Yaskawa INFORM job: u_tourne4TRJ0.JBI

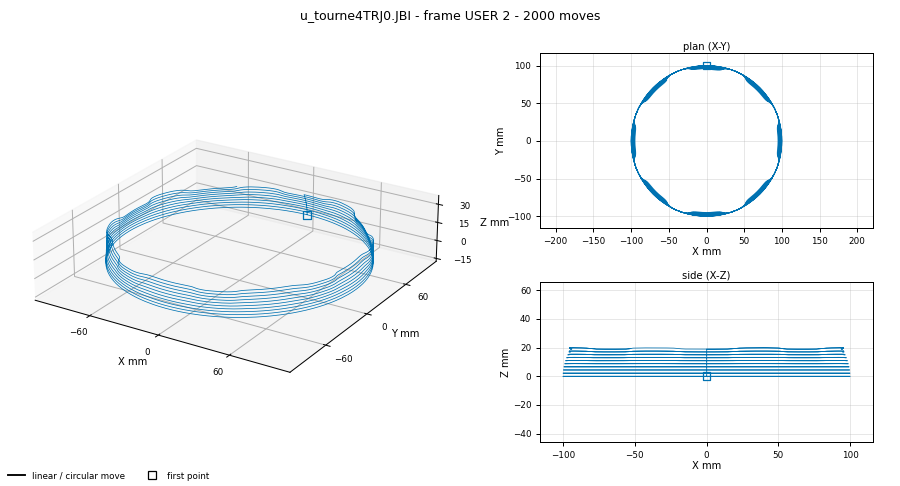
[picture p0: tool path of u_tourne4TRJ0.JBI in frame USER 2, 2000 of 2000 moves have a stored position in this frame; points joined in program order, loops and branches not executed]
/JOB
//NAME u_tourne4TRJ0
///FOLDERNAME DEMO
//POS
///NPOS 2000,0,2000,0,0,0
///USER 2
///TOOL 7
///POSTYPE USER
///RECTAN
///RCONF 1,0,0,0,0,0,0,0,0,0,0,0,0,0,0,0,0,0,0,0,0,0,0,0
C00000=0.000,100.000,0.000,-180.0000,0.0000,-90.0000
C00001=5.792,99.832,0.000,-180.0000,0.0000,-93.3204
C00002=10.988,99.394,0.000,-180.0000,0.0000,-96.3084
C00003=15.564,98.781,0.000,-180.0000,0.0000,-98.9540
C00004=18.698,98.237,0.000,-180.0000,0.0000,-100.7765
C00005=20.854,97.801,0.000,-180.0000,0.0000,-102.0369
C00006=22.593,97.414,0.000,-180.0000,0.0000,-103.0576
C00007=24.351,96.990,0.000,-180.0000,0.0000,-104.0938
C00008=26.550,96.411,0.000,-180.0000,0.0000,-105.3967
C00009=29.248,95.627,0.000,-180.0000,0.0000,-107.0065
C00010=32.094,94.710,0.000,-180.0000,0.0000,-108.7198
C00011=34.739,93.772,0.000,-180.0000,0.0000,-110.3278
C00012=37.121,92.855,0.000,-180.0000,0.0000,-111.7902
C00013=39.410,91.907,0.000,-180.0000,0.0000,-113.2098
C00014=41.743,90.871,0.000,-180.0000,0.0000,-114.6724
C00015=44.276,89.664,0.000,-180.0000,-0.0000,-116.2801
C00016=46.937,88.300,0.000,-180.0000,-0.0000,-117.9935
C00017=49.400,86.946,0.000,-180.0000,0.0000,-119.6039
C00018=51.363,85.801,0.000,-180.0000,0.0000,-120.9060
C00019=52.906,84.858,0.000,-180.0000,0.0000,-121.9421
C00020=54.410,83.902,0.000,-180.0000,0.0000,-122.9632
C00021=56.242,82.685,0.000,-180.0000,0.0000,-124.2234
C00022=58.844,80.854,0.000,-180.0000,0.0000,-126.0464
C00023=62.512,78.053,0.000,-180.0000,0.0000,-128.6909
C00024=66.496,74.687,0.000,-180.0000,0.0000,-131.6796
C00025=70.711,70.711,0.000,-180.0000,0.0000,-135.0000
C00026=74.687,66.496,0.000,-180.0000,0.0000,-138.3204
C00027=78.053,62.512,0.000,-180.0000,0.0000,-141.3091
C00028=80.854,58.844,0.000,-180.0000,-0.0000,-143.9536
C00029=82.685,56.242,0.000,-180.0000,0.0000,-145.7766
C00030=83.902,54.410,0.000,-180.0000,0.0000,-147.0368
C00031=84.858,52.906,0.000,-180.0000,0.0000,-148.0579
C00032=85.801,51.363,0.000,-180.0000,0.0000,-149.0940
C00033=86.946,49.400,0.000,-180.0000,0.0000,-150.3961
C00034=88.300,46.937,0.000,-180.0000,0.0000,-152.0065
C00035=89.664,44.276,0.000,-180.0000,0.0000,-153.7199
C00036=90.871,41.743,0.000,-180.0000,0.0000,-155.3276
C00037=91.907,39.410,0.000,-180.0000,0.0000,-156.7902
C00038=92.855,37.121,0.000,-180.0000,0.0000,-158.2098
C00039=93.772,34.739,0.000,-180.0000,0.0000,-159.6722
C00040=94.710,32.094,0.000,-180.0000,0.0000,-161.2802
C00041=95.627,29.248,0.000,-180.0000,0.0000,-162.9935
C00042=96.411,26.550,0.000,-180.0000,0.0000,-164.6033
C00043=96.990,24.351,0.000,-180.0000,0.0000,-165.9062
C00044=97.414,22.593,0.000,-180.0000,0.0000,-166.9424
C00045=97.801,20.854,0.000,-180.0000,0.0000,-167.9631
C00046=98.237,18.698,0.000,-180.0000,0.0000,-169.2235
C00047=98.781,15.564,0.000,-180.0000,0.0000,-171.0460
C00048=99.394,10.988,0.000,-180.0000,0.0000,-173.6916
C00049=99.832,5.792,0.000,-180.0000,0.0000,-176.6796
C00050=100.000,0.000,0.000,-180.0000,0.0000,-180.0000
C00051=99.832,-5.792,0.000,-180.0000,0.0000,-183.3204
C00052=99.394,-10.988,0.000,-180.0000,0.0000,-186.3084
C00053=98.781,-15.564,0.000,-180.0000,0.0000,-188.9540
C00054=98.237,-18.698,0.000,-180.0000,0.0000,-190.7765
C00055=97.801,-20.854,0.000,-180.0000,0.0000,-192.0369
C00056=97.414,-22.593,0.000,-180.0000,0.0000,-193.0576
C00057=96.990,-24.351,0.000,-180.0000,0.0000,-194.0938
C00058=96.411,-26.550,0.000,-180.0000,0.0000,-195.3967
C00059=95.627,-29.248,0.000,-180.0000,0.0000,-197.0065
C00060=94.710,-32.094,0.000,-180.0000,0.0000,-198.7198
C00061=93.772,-34.739,0.000,-180.0000,0.0000,-200.3278
C00062=92.855,-37.121,0.000,-180.0000,0.0000,-201.7902
C00063=91.907,-39.410,0.000,-180.0000,0.0000,-203.2098
C00064=90.871,-41.743,0.000,-180.0000,0.0000,-204.6724
C00065=89.664,-44.276,0.000,-180.0000,0.0000,-206.2801
C00066=88.300,-46.937,0.000,-180.0000,0.0000,-207.9935
C00067=86.946,-49.400,0.000,-180.0000,0.0000,-209.6039
C00068=85.801,-51.363,0.000,-180.0000,0.0000,-210.9060
C00069=84.858,-52.906,0.000,-180.0000,0.0000,-211.9421
C00070=83.902,-54.410,0.000,-180.0000,0.0000,-212.9632
C00071=82.685,-56.242,0.000,-180.0000,0.0000,-214.2234
C00072=80.854,-58.844,0.000,-180.0000,0.0000,-216.0464
C00073=78.053,-62.512,0.000,-180.0000,0.0000,-218.6909
C00074=74.687,-66.496,0.000,-180.0000,0.0000,-221.6796
C00075=70.711,-70.711,0.000,-180.0000,0.0000,-225.0000
C00076=66.496,-74.687,0.000,-180.0000,0.0000,-228.3204
C00077=62.512,-78.053,0.000,-180.0000,0.0000,-231.3091
C00078=58.844,-80.854,0.000,-180.0000,0.0000,-233.9536
C00079=56.242,-82.685,0.000,-180.0000,0.0000,-235.7766
C00080=54.410,-83.902,0.000,-180.0000,0.0000,-237.0368
C00081=52.906,-84.858,0.000,-180.0000,0.0000,-238.0579
C00082=51.363,-85.801,0.000,-180.0000,0.0000,-239.0940
C00083=49.400,-86.946,0.000,-180.0000,-0.0000,-240.3961
C00084=46.937,-88.300,0.000,-180.0000,0.0000,-242.0065
C00085=44.276,-89.664,0.000,-180.0000,0.0000,-243.7199
C00086=41.743,-90.871,0.000,-180.0000,0.0000,-245.3276
C00087=39.410,-91.907,0.000,-180.0000,0.0000,-246.7902
C00088=37.121,-92.855,0.000,-180.0000,0.0000,-248.2098
C00089=34.739,-93.772,0.000,-180.0000,0.0000,-249.6722
C00090=32.094,-94.710,0.000,-180.0000,0.0000,-251.2802
C00091=29.248,-95.627,0.000,-180.0000,0.0000,-252.9935
C00092=26.550,-96.411,0.000,-180.0000,0.0000,-254.6033
C00093=24.351,-96.990,0.000,-180.0000,0.0000,-255.9062
C00094=22.593,-97.414,0.000,-180.0000,0.0000,-256.9424
C00095=20.854,-97.801,0.000,-180.0000,0.0000,-257.9631
C00096=18.698,-98.237,0.000,-180.0000,0.0000,-259.2235
C00097=15.564,-98.781,0.000,-180.0000,0.0000,-261.0460
C00098=10.988,-99.394,0.000,-180.0000,0.0000,-263.6916
C00099=5.792,-99.832,0.000,-180.0000,0.0000,-266.6796
C00100=0.000,-100.000,0.000,180.0000,-0.0000,-270.0000
C00101=0.000,-100.000,0.000,180.0000,-0.0000,-270.0000
C00102=-5.792,-99.832,0.000,-180.0000,-0.0000,-273.3204
C00103=-10.988,-99.394,0.000,-180.0000,-0.0000,-276.3084
C00104=-15.564,-98.781,0.000,-180.0000,-0.0000,-278.9540
C00105=-18.698,-98.237,0.000,-180.0000,-0.0000,-280.7765
C00106=-20.854,-97.801,0.000,-180.0000,-0.0000,-282.0369
C00107=-22.593,-97.414,0.000,-180.0000,-0.0000,-283.0576
C00108=-24.351,-96.990,0.000,-180.0000,-0.0000,-284.0938
C00109=-26.550,-96.411,0.000,-180.0000,-0.0000,-285.3967
C00110=-29.248,-95.627,0.000,-180.0000,-0.0000,-287.0065
C00111=-32.094,-94.710,0.000,-180.0000,-0.0000,-288.7198
C00112=-34.739,-93.772,0.000,-180.0000,-0.0000,-290.3278
C00113=-37.121,-92.855,0.000,-180.0000,-0.0000,-291.7902
C00114=-39.410,-91.907,0.000,-180.0000,-0.0000,-293.2098
C00115=-41.743,-90.871,0.000,-180.0000,-0.0000,-294.6724
C00116=-44.276,-89.664,0.000,-180.0000,-0.0000,-296.2801
C00117=-46.937,-88.300,0.000,-180.0000,-0.0000,-297.9935
C00118=-49.400,-86.946,0.000,-180.0000,-0.0000,-299.6039
C00119=-51.363,-85.801,0.000,-180.0000,-0.0000,-300.9060
C00120=-52.906,-84.858,0.000,-180.0000,-0.0000,-301.9421
C00121=-54.410,-83.902,0.000,-180.0000,-0.0000,-302.9632
C00122=-56.242,-82.685,0.000,-180.0000,-0.0000,-304.2234
C00123=-58.844,-80.854,0.000,-180.0000,-0.0000,-306.0464
C00124=-62.512,-78.053,0.000,-180.0000,-0.0000,-308.6909
C00125=-66.496,-74.687,0.000,-180.0000,-0.0000,-311.6796
C00126=-70.711,-70.711,0.000,-180.0000,-0.0000,-315.0000
C00127=-74.687,-66.496,0.000,-180.0000,-0.0000,-318.3204
C00128=-78.053,-62.512,0.000,-180.0000,-0.0000,-321.3091
C00129=-80.854,-58.844,0.000,-180.0000,-0.0000,-323.9536
C00130=-82.685,-56.242,0.000,-180.0000,-0.0000,-325.7766
C00131=-83.902,-54.410,0.000,-180.0000,-0.0000,-327.0368
C00132=-84.858,-52.906,0.000,-180.0000,-0.0000,-328.0579
C00133=-85.801,-51.363,0.000,-180.0000,-0.0000,-329.0940
C00134=-86.946,-49.400,0.000,-180.0000,-0.0000,-330.3961
C00135=-88.300,-46.937,0.000,-180.0000,-0.0000,-332.0065
C00136=-89.664,-44.276,0.000,-180.0000,-0.0000,-333.7199
C00137=-90.871,-41.743,0.000,-180.0000,0.0000,-335.3276
C00138=-91.907,-39.410,0.000,-180.0000,0.0000,-336.7902
C00139=-92.855,-37.121,0.000,-180.0000,-0.0000,-338.2098
C00140=-93.772,-34.739,0.000,-180.0000,-0.0000,-339.6722
C00141=-94.710,-32.094,0.000,-180.0000,0.0000,-341.2802
C00142=-95.627,-29.248,0.000,-180.0000,0.0000,-342.9935
C00143=-96.411,-26.550,0.000,-180.0000,-0.0000,-344.6033
C00144=-96.990,-24.351,0.000,-180.0000,-0.0000,-345.9062
C00145=-97.414,-22.593,0.000,-180.0000,-0.0000,-346.9424
C00146=-97.801,-20.854,0.000,-180.0000,-0.0000,-347.9631
C00147=-98.237,-18.698,0.000,-180.0000,-0.0000,-349.2235
C00148=-98.781,-15.564,0.000,-180.0000,-0.0000,-351.0460
C00149=-99.394,-10.988,0.000,-180.0000,-0.0000,-353.6916
C00150=-99.832,-5.792,0.000,-180.0000,-0.0000,-356.6796
C00151=-100.000,0.000,0.000,-180.0000,0.0000,-360.0000
C00152=-99.832,5.792,0.000,-180.0000,0.0000,-363.3204
C00153=-99.394,10.988,0.000,-180.0000,0.0000,-366.3084
C00154=-98.781,15.564,0.000,-180.0000,0.0000,-368.9540
C00155=-98.237,18.698,0.000,-180.0000,0.0000,-370.7765
C00156=-97.801,20.854,0.000,-180.0000,0.0000,-372.0369
C00157=-97.414,22.593,0.000,-180.0000,0.0000,-373.0576
C00158=-96.990,24.351,0.000,-180.0000,0.0000,-374.0938
C00159=-96.411,26.550,0.000,-180.0000,0.0000,-375.3967
C00160=-95.627,29.248,0.000,-180.0000,0.0000,-377.0065
C00161=-94.710,32.094,0.000,-180.0000,0.0000,-378.7198
C00162=-93.772,34.739,0.000,-180.0000,0.0000,-380.3278
C00163=-92.855,37.121,0.000,-180.0000,0.0000,-381.7902
C00164=-91.907,39.410,0.000,-180.0000,0.0000,-383.2098
C00165=-90.871,41.743,0.000,-180.0000,0.0000,-384.6724
C00166=-89.664,44.276,0.000,-180.0000,0.0000,-386.2801
C00167=-88.300,46.937,0.000,-180.0000,0.0000,-387.9935
C00168=-86.946,49.400,0.000,-180.0000,0.0000,-389.6039
C00169=-85.801,51.363,0.000,-180.0000,0.0000,-390.9060
C00170=-84.858,52.906,0.000,-180.0000,0.0000,-391.9421
C00171=-83.902,54.410,0.000,-180.0000,0.0000,-392.9632
C00172=-82.685,56.242,0.000,-180.0000,0.0000,-394.2234
C00173=-80.854,58.844,0.000,-180.0000,0.0000,-396.0464
C00174=-78.053,62.512,0.000,-180.0000,0.0000,-398.6909
C00175=-74.687,66.496,0.000,-180.0000,0.0000,-401.6796
C00176=-70.711,70.711,0.000,-180.0000,0.0000,-405.0000
C00177=-66.496,74.687,0.000,-180.0000,0.0000,-408.3204
C00178=-62.512,78.053,0.000,-180.0000,0.0000,-411.3091
C00179=-58.844,80.854,0.000,-180.0000,0.0000,-413.9536
C00180=-56.242,82.685,0.000,-180.0000,0.0000,-415.7766
C00181=-54.410,83.902,0.000,-180.0000,0.0000,-417.0368
C00182=-52.906,84.858,0.000,-180.0000,0.0000,-418.0579
C00183=-51.363,85.801,0.000,-180.0000,0.0000,-419.0940
C00184=-49.400,86.946,0.000,-180.0000,0.0000,-420.3961
C00185=-46.937,88.300,0.000,-180.0000,0.0000,-422.0065
C00186=-44.276,89.664,0.000,-180.0000,0.0000,-423.7199
C00187=-41.743,90.871,0.000,-180.0000,0.0000,-425.3276
C00188=-39.410,91.907,0.000,-180.0000,0.0000,-426.7902
C00189=-37.121,92.855,0.000,-180.0000,0.0000,-428.2098
C00190=-34.739,93.772,0.000,-180.0000,0.0000,-429.6722
C00191=-32.094,94.710,0.000,-180.0000,0.0000,-431.2802
C00192=-29.248,95.627,0.000,-180.0000,0.0000,-432.9935
C00193=-26.550,96.411,0.000,-180.0000,0.0000,-434.6033
C00194=-24.351,96.990,0.000,-180.0000,0.0000,-435.9062
C00195=-22.593,97.414,0.000,-180.0000,0.0000,-436.9424
C00196=-20.854,97.801,0.000,-180.0000,0.0000,-437.9631
C00197=-18.698,98.237,0.000,-180.0000,0.0000,-439.2235
C00198=-15.564,98.781,0.000,-180.0000,0.0000,-441.0460
C00199=-10.988,99.394,0.000,-180.0000,0.0000,-443.6916
C00200=-5.792,99.832,0.000,-180.0000,0.0000,-446.6796
C00201=0.000,100.000,0.000,-180.0000,0.0000,-450.0000
C00202=0.000,99.921,2.199,-180.0000,4.0599,-450.0000
C00203=5.785,99.754,2.199,180.0000,4.0610,-453.3190
C00204=10.976,99.317,2.199,-179.9982,4.0560,-456.3064
C00205=15.549,98.707,2.199,179.9951,3.8999,-458.9521
C00206=18.681,98.171,2.199,179.9877,3.4994,-460.7740
C00207=20.835,97.748,2.199,179.9835,2.9093,-462.0325
C00208=22.573,97.375,2.200,179.9797,2.2192,-463.0515
C00209=24.330,96.965,2.200,179.9890,1.5274,-464.0856
C00210=26.527,96.399,2.200,179.9949,0.9256,-465.3858
C00211=29.226,95.625,2.200,-179.9996,0.4495,-466.9948
C00212=32.077,94.713,2.200,179.9994,0.1268,-468.7100
C00213=34.728,93.776,2.200,179.9994,0.0181,-470.3211
C00214=37.118,92.856,2.200,-180.0000,0.0000,-471.7884
C00215=39.413,91.905,2.200,-180.0000,0.0000,-473.2118
C00216=41.753,90.866,2.200,-179.9968,0.0204,-474.6788
C00217=44.291,89.654,2.200,-179.9994,0.1281,-476.2904
C00218=46.951,88.283,2.200,-179.9985,0.4486,-478.0051
C00219=49.407,86.922,2.200,-179.9929,0.9267,-479.6142
C00220=51.360,85.768,2.200,-179.9928,1.5272,-480.9142
C00221=52.893,84.816,2.200,-179.9802,2.2211,-481.9485
C00222=54.385,83.851,2.199,-179.9808,2.9093,-482.9671
C00223=56.208,82.627,2.199,-179.9866,3.4970,-484.2260
C00224=58.802,80.791,2.199,-179.9934,3.8982,-486.0482
C00225=62.466,77.989,2.199,179.9994,4.0551,-488.6933
C00226=66.446,74.627,2.199,180.0000,4.0616,-491.6811
C00227=70.655,70.655,2.199,180.0000,4.0629,-495.0000
C00228=74.627,66.446,2.199,-180.0000,4.0616,-498.3189
C00229=77.989,62.466,2.199,-179.9994,4.0551,-501.3067
C00230=80.791,58.802,2.199,179.9934,3.8982,-503.9518
C00231=82.627,56.208,2.199,179.9866,3.4970,-505.7740
C00232=83.851,54.385,2.199,179.9808,2.9093,-507.0329
C00233=84.816,52.893,2.200,179.9802,2.2211,-508.0515
C00234=85.768,51.360,2.200,179.9928,1.5272,-509.0858
C00235=86.922,49.407,2.200,179.9929,0.9267,-510.3858
C00236=88.283,46.951,2.200,179.9985,0.4486,-511.9949
C00237=89.654,44.291,2.200,179.9994,0.1281,-513.7096
C00238=90.866,41.753,2.200,179.9968,0.0204,-515.3212
C00239=91.905,39.413,2.200,-180.0000,0.0000,-516.7882
C00240=92.856,37.118,2.200,-180.0000,0.0000,-518.2116
C00241=93.776,34.728,2.200,-179.9994,0.0181,-519.6789
C00242=94.713,32.077,2.200,-179.9994,0.1268,-521.2900
C00243=95.625,29.226,2.200,179.9996,0.4495,-523.0052
C00244=96.399,26.527,2.200,-179.9949,0.9256,-524.6142
C00245=96.965,24.330,2.200,-179.9890,1.5274,-525.9144
C00246=97.375,22.573,2.200,-179.9797,2.2192,-526.9485
C00247=97.748,20.835,2.199,-179.9835,2.9093,-527.9675
C00248=98.171,18.681,2.199,-179.9877,3.4994,-529.2260
C00249=98.707,15.549,2.199,-179.9951,3.8999,-531.0479
C00250=99.317,10.976,2.199,179.9982,4.0560,-533.6936
C00251=99.754,5.785,2.199,-180.0000,4.0610,-536.6810
C00252=99.921,0.000,2.199,-180.0000,4.0599,-540.0000
C00253=99.754,-5.785,2.199,180.0000,4.0610,-543.3190
C00254=99.317,-10.976,2.199,-179.9982,4.0560,-546.3064
C00255=98.707,-15.549,2.199,179.9951,3.8999,-548.9521
C00256=98.171,-18.681,2.199,179.9877,3.4994,-550.7740
C00257=97.748,-20.835,2.199,179.9835,2.9093,-552.0325
C00258=97.375,-22.573,2.200,179.9797,2.2192,-553.0515
C00259=96.965,-24.330,2.200,179.9890,1.5274,-554.0856
C00260=96.399,-26.527,2.200,179.9949,0.9256,-555.3858
C00261=95.625,-29.226,2.200,-179.9996,0.4495,-556.9948
C00262=94.713,-32.077,2.200,179.9994,0.1268,-558.7100
C00263=93.776,-34.728,2.200,179.9994,0.0181,-560.3211
C00264=92.856,-37.118,2.200,-180.0000,0.0000,-561.7884
C00265=91.905,-39.413,2.200,-180.0000,0.0000,-563.2118
C00266=90.866,-41.753,2.200,-179.9968,0.0204,-564.6788
C00267=89.654,-44.291,2.200,-179.9994,0.1281,-566.2904
C00268=88.283,-46.951,2.200,-179.9985,0.4486,-568.0051
C00269=86.922,-49.407,2.200,-179.9929,0.9267,-569.6142
C00270=85.768,-51.360,2.200,-179.9928,1.5272,-570.9142
C00271=84.816,-52.893,2.200,-179.9802,2.2211,-571.9485
C00272=83.851,-54.385,2.199,-179.9808,2.9093,-572.9671
C00273=82.627,-56.208,2.199,-179.9866,3.4970,-574.2260
C00274=80.791,-58.802,2.199,-179.9934,3.8982,-576.0482
C00275=77.989,-62.466,2.199,179.9994,4.0551,-578.6933
C00276=74.627,-66.446,2.199,180.0000,4.0616,-581.6811
C00277=70.655,-70.655,2.199,180.0000,4.0629,-585.0000
C00278=66.446,-74.627,2.199,-180.0000,4.0616,-588.3189
C00279=62.466,-77.989,2.199,-179.9994,4.0551,-591.3067
C00280=58.802,-80.791,2.199,179.9934,3.8982,-593.9518
C00281=56.208,-82.627,2.199,179.9866,3.4970,-595.7740
C00282=54.385,-83.851,2.199,179.9808,2.9093,-597.0329
C00283=52.893,-84.816,2.200,179.9802,2.2211,-598.0515
C00284=51.360,-85.768,2.200,179.9928,1.5272,-599.0858
C00285=49.407,-86.922,2.200,179.9929,0.9267,-600.3858
C00286=46.951,-88.283,2.200,179.9985,0.4486,-601.9949
C00287=44.291,-89.654,2.200,179.9994,0.1281,-603.7096
C00288=41.753,-90.866,2.200,179.9968,0.0204,-605.3212
C00289=39.413,-91.905,2.200,-180.0000,0.0000,-606.7882
C00290=37.118,-92.856,2.200,-180.0000,0.0000,-608.2116
C00291=34.728,-93.776,2.200,-179.9994,0.0181,-609.6789
C00292=32.077,-94.713,2.200,-179.9994,0.1268,-611.2900
C00293=29.226,-95.625,2.200,179.9996,0.4495,-613.0052
C00294=26.527,-96.399,2.200,-179.9949,0.9256,-614.6142
C00295=24.330,-96.965,2.200,-179.9890,1.5274,-615.9144
C00296=22.573,-97.375,2.200,-179.9797,2.2192,-616.9485
C00297=20.835,-97.748,2.199,-179.9835,2.9093,-617.9675
C00298=18.681,-98.171,2.199,-179.9877,3.4994,-619.2260
C00299=15.549,-98.707,2.199,-179.9951,3.8999,-621.0479
C00300=10.976,-99.317,2.199,179.9982,4.0560,-623.6936
C00301=5.785,-99.754,2.199,-180.0000,4.0610,-626.6810
C00302=0.000,-99.921,2.199,-180.0000,4.0599,-630.0000
C00303=0.000,-99.921,2.199,-180.0000,4.0599,-630.0000
C00304=-5.785,-99.754,2.199,180.0000,4.0610,-633.3190
C00305=-10.976,-99.317,2.199,-179.9982,4.0560,-636.3064
C00306=-15.549,-98.707,2.199,179.9951,3.8999,-638.9521
C00307=-18.681,-98.171,2.199,179.9877,3.4994,-640.7740
C00308=-20.835,-97.748,2.199,179.9835,2.9093,-642.0325
C00309=-22.573,-97.375,2.200,179.9797,2.2192,-643.0515
C00310=-24.330,-96.965,2.200,179.9890,1.5274,-644.0856
C00311=-26.527,-96.399,2.200,179.9949,0.9256,-645.3858
C00312=-29.226,-95.625,2.200,-179.9996,0.4495,-646.9948
C00313=-32.077,-94.713,2.200,179.9994,0.1268,-648.7100
C00314=-34.728,-93.776,2.200,179.9994,0.0181,-650.3211
C00315=-37.118,-92.856,2.200,-180.0000,0.0000,-651.7884
C00316=-39.413,-91.905,2.200,-180.0000,0.0000,-653.2118
C00317=-41.753,-90.866,2.200,-179.9968,0.0204,-654.6788
C00318=-44.291,-89.654,2.200,-179.9994,0.1281,-656.2904
C00319=-46.951,-88.283,2.200,-179.9985,0.4486,-658.0051
C00320=-49.407,-86.922,2.200,-179.9929,0.9267,-659.6142
C00321=-51.360,-85.768,2.200,-179.9928,1.5272,-660.9142
C00322=-52.893,-84.816,2.200,-179.9802,2.2211,-661.9485
C00323=-54.385,-83.851,2.199,-179.9808,2.9093,-662.9671
C00324=-56.208,-82.627,2.199,-179.9866,3.4970,-664.2260
C00325=-58.802,-80.791,2.199,-179.9934,3.8982,-666.0482
C00326=-62.466,-77.989,2.199,179.9994,4.0551,-668.6933
C00327=-66.446,-74.627,2.199,180.0000,4.0616,-671.6811
C00328=-70.655,-70.655,2.199,180.0000,4.0629,-675.0000
C00329=-74.627,-66.446,2.199,-180.0000,4.0616,-678.3189
C00330=-77.989,-62.466,2.199,-179.9994,4.0551,-681.3067
C00331=-80.791,-58.802,2.199,179.9934,3.8982,-683.9518
C00332=-82.627,-56.208,2.199,179.9866,3.4970,-685.7740
C00333=-83.851,-54.385,2.199,179.9808,2.9093,-687.0329
C00334=-84.816,-52.893,2.200,179.9802,2.2211,-688.0515
C00335=-85.768,-51.360,2.200,179.9928,1.5272,-689.0858
C00336=-86.922,-49.407,2.200,179.9929,0.9267,-690.3858
C00337=-88.283,-46.951,2.200,179.9985,0.4486,-691.9949
C00338=-89.654,-44.291,2.200,179.9994,0.1281,-693.7096
C00339=-90.866,-41.753,2.200,179.9968,0.0204,-695.3212
C00340=-91.905,-39.413,2.200,-180.0000,0.0000,-696.7882
C00341=-92.856,-37.118,2.200,-180.0000,0.0000,-698.2116
C00342=-93.776,-34.728,2.200,-179.9994,0.0181,-699.6789
C00343=-94.713,-32.077,2.200,-179.9994,0.1268,-701.2900
C00344=-95.625,-29.226,2.200,179.9996,0.4495,-703.0052
C00345=-96.399,-26.527,2.200,-179.9949,0.9256,-704.6142
C00346=-96.965,-24.330,2.200,-179.9890,1.5274,-705.9144
C00347=-97.375,-22.573,2.200,-179.9797,2.2192,-706.9485
C00348=-97.748,-20.835,2.199,-179.9835,2.9093,-707.9675
C00349=-98.171,-18.681,2.199,-179.9877,3.4994,-709.2260
C00350=-98.707,-15.549,2.199,-179.9951,3.8999,-711.0479
C00351=-99.317,-10.976,2.199,179.9982,4.0560,-713.6936
C00352=-99.754,-5.785,2.199,-180.0000,4.0610,-716.6810
C00353=-99.921,0.000,2.199,-180.0000,4.0599,-720.0000
C00354=-99.754,5.785,2.199,180.0000,4.0610,-723.3190
C00355=-99.317,10.976,2.199,-179.9982,4.0560,-726.3064
C00356=-98.707,15.549,2.199,179.9951,3.8999,-728.9521
C00357=-98.171,18.681,2.199,179.9877,3.4994,-730.7740
C00358=-97.748,20.835,2.199,179.9835,2.9093,-732.0325
C00359=-97.375,22.573,2.200,179.9797,2.2192,-733.0515
C00360=-96.965,24.330,2.200,179.9890,1.5274,-734.0856
C00361=-96.399,26.527,2.200,179.9949,0.9256,-735.3858
C00362=-95.625,29.226,2.200,-179.9996,0.4495,-736.9948
C00363=-94.713,32.077,2.200,179.9994,0.1268,-738.7100
C00364=-93.776,34.728,2.200,179.9994,0.0181,-740.3211
C00365=-92.856,37.118,2.200,-180.0000,0.0000,-741.7884
C00366=-91.905,39.413,2.200,-180.0000,0.0000,-743.2118
C00367=-90.866,41.753,2.200,-179.9968,0.0204,-744.6788
C00368=-89.654,44.291,2.200,-179.9994,0.1281,-746.2904
C00369=-88.283,46.951,2.200,-179.9985,0.4486,-748.0051
C00370=-86.922,49.407,2.200,-179.9929,0.9267,-749.6142
C00371=-85.768,51.360,2.200,-179.9928,1.5272,-750.9142
C00372=-84.816,52.893,2.200,-179.9802,2.2211,-751.9485
C00373=-83.851,54.385,2.199,-179.9808,2.9093,-752.9671
C00374=-82.627,56.208,2.199,-179.9866,3.4970,-754.2260
C00375=-80.791,58.802,2.199,-179.9934,3.8982,-756.0482
C00376=-77.989,62.466,2.199,179.9994,4.0551,-758.6933
C00377=-74.627,66.446,2.199,180.0000,4.0616,-761.6811
C00378=-70.655,70.655,2.199,180.0000,4.0629,-765.0000
C00379=-66.446,74.627,2.199,-180.0000,4.0616,-768.3189
C00380=-62.466,77.989,2.199,-179.9994,4.0551,-771.3067
C00381=-58.802,80.791,2.199,179.9934,3.8982,-773.9518
C00382=-56.208,82.627,2.199,179.9866,3.4970,-775.7740
C00383=-54.385,83.851,2.199,179.9808,2.9093,-777.0329
C00384=-52.893,84.816,2.200,179.9802,2.2211,-778.0515
C00385=-51.360,85.768,2.200,179.9928,1.5272,-779.0858
C00386=-49.407,86.922,2.200,179.9929,0.9267,-780.3858
C00387=-46.951,88.283,2.200,179.9985,0.4486,-781.9949
C00388=-44.291,89.654,2.200,179.9994,0.1281,-783.7096
C00389=-41.753,90.866,2.200,179.9968,0.0204,-785.3212
C00390=-39.413,91.905,2.200,-180.0000,0.0000,-786.7882
C00391=-37.118,92.856,2.200,-180.0000,0.0000,-788.2116
C00392=-34.728,93.776,2.200,-179.9994,0.0181,-789.6789
C00393=-32.077,94.713,2.200,-179.9994,0.1268,-791.2900
C00394=-29.226,95.625,2.200,179.9996,0.4495,-793.0052
C00395=-26.527,96.399,2.200,-179.9949,0.9256,-794.6142
C00396=-24.330,96.965,2.200,-179.9890,1.5274,-795.9144
C00397=-22.573,97.375,2.200,-179.9797,2.2192,-796.9485
C00398=-20.835,97.748,2.199,-179.9835,2.9093,-797.9675
C00399=-18.681,98.171,2.199,-179.9877,3.4994,-799.2260
C00400=-15.549,98.707,2.199,-179.9951,3.8999,-801.0479
C00401=-10.976,99.317,2.199,179.9982,4.0560,-803.6936
C00402=-5.785,99.754,2.199,-180.0000,4.0610,-806.6810
C00403=0.000,99.921,2.199,-180.0000,4.0599,-810.0000
C00404=0.000,99.691,4.387,-180.0000,7.8975,-810.0000
C00405=5.764,99.524,4.387,-179.9969,7.8994,-813.3146
C00406=10.941,99.090,4.387,179.9908,7.8868,-816.3008
C00407=15.506,98.490,4.388,179.9574,7.5851,-818.9471
C00408=18.630,97.979,4.390,179.8975,6.8083,-820.7659
C00409=20.779,97.591,4.393,179.8518,5.6544,-822.0199
C00410=22.514,97.259,4.396,179.8623,4.3065,-823.0335
C00411=24.268,96.890,4.398,179.9222,2.9528,-824.0616
C00412=26.460,96.362,4.399,179.9728,1.7872,-825.3544
C00413=29.164,95.617,4.399,179.9911,0.8539,-826.9622
C00414=32.027,94.722,4.399,179.9972,0.2410,-828.6812
C00415=34.697,93.786,4.400,179.9988,0.0362,-830.3024
C00416=37.107,92.860,4.400,179.9979,0.0053,-831.7817
C00417=39.424,91.901,4.400,179.9977,0.0053,-833.2185
C00418=41.782,90.851,4.400,-179.9987,0.0384,-834.6975
C00419=44.332,89.625,4.399,-179.9990,0.2434,-836.3188
C00420=46.990,88.233,4.399,-179.9887,0.8564,-838.0383
C00421=49.428,86.848,4.399,-179.9706,1.7904,-839.6456
C00422=51.352,85.672,4.398,-179.9249,2.9520,-840.9386
C00423=52.853,84.692,4.396,-179.8607,4.3050,-841.9667
C00424=54.314,83.700,4.393,-179.8530,5.6572,-842.9801
C00425=56.108,82.455,4.390,-179.8953,6.8088,-844.2340
C00426=58.679,80.608,4.388,-179.9571,7.5869,-846.0529
C00427=62.331,77.804,4.387,-179.9919,7.8870,-848.6992
C00428=66.299,74.450,4.387,179.9976,7.9022,-851.6856
C00429=70.493,70.493,4.387,180.0000,7.9010,-855.0000
C00430=74.450,66.299,4.387,-179.9976,7.9022,-858.3144
C00431=77.804,62.331,4.387,179.9919,7.8870,-861.3008
C00432=80.608,58.679,4.388,179.9571,7.5869,-863.9471
C00433=82.455,56.108,4.390,179.8953,6.8088,-865.7660
C00434=83.700,54.314,4.393,179.8530,5.6572,-867.0199
C00435=84.692,52.853,4.396,179.8607,4.3050,-868.0333
C00436=85.672,51.352,4.398,179.9249,2.9520,-869.0614
C00437=86.848,49.428,4.399,179.9706,1.7904,-870.3544
C00438=88.233,46.990,4.399,179.9887,0.8564,-871.9617
C00439=89.625,44.332,4.399,179.9990,0.2434,-873.6812
C00440=90.851,41.782,4.400,179.9987,0.0384,-875.3025
C00441=91.901,39.424,4.400,-179.9977,0.0053,-876.7815
C00442=92.860,37.107,4.400,-179.9979,0.0053,-878.2183
C00443=93.786,34.697,4.400,-179.9988,0.0362,-879.6976
C00444=94.722,32.027,4.399,-179.9972,0.2410,-881.3188
C00445=95.617,29.164,4.399,-179.9911,0.8539,-883.0378
C00446=96.362,26.460,4.399,-179.9728,1.7872,-884.6456
C00447=96.890,24.268,4.398,-179.9222,2.9528,-885.9384
C00448=97.259,22.514,4.396,-179.8623,4.3065,-886.9665
C00449=97.591,20.779,4.393,-179.8518,5.6544,-887.9801
C00450=97.979,18.630,4.390,-179.8975,6.8083,-889.2341
C00451=98.490,15.506,4.388,-179.9574,7.5851,-891.0529
C00452=99.090,10.941,4.387,-179.9908,7.8868,-893.6992
C00453=99.524,5.764,4.387,179.9969,7.8994,-896.6854
C00454=99.691,0.000,4.387,-180.0000,7.8975,-900.0000
C00455=99.524,-5.764,4.387,-179.9969,7.8994,-903.3146
C00456=99.090,-10.941,4.387,179.9908,7.8868,-906.3008
C00457=98.490,-15.506,4.388,179.9574,7.5851,-908.9471
C00458=97.979,-18.630,4.390,179.8975,6.8083,-910.7659
C00459=97.591,-20.779,4.393,179.8518,5.6544,-912.0199
C00460=97.259,-22.514,4.396,179.8623,4.3065,-913.0335
C00461=96.890,-24.268,4.398,179.9222,2.9528,-914.0616
C00462=96.362,-26.460,4.399,179.9728,1.7872,-915.3544
C00463=95.617,-29.164,4.399,179.9911,0.8539,-916.9622
C00464=94.722,-32.027,4.399,179.9972,0.2410,-918.6812
C00465=93.786,-34.697,4.400,179.9988,0.0362,-920.3024
C00466=92.860,-37.107,4.400,179.9979,0.0053,-921.7817
C00467=91.901,-39.424,4.400,179.9977,0.0053,-923.2185
C00468=90.851,-41.782,4.400,-179.9987,0.0384,-924.6975
C00469=89.625,-44.332,4.399,-179.9990,0.2434,-926.3188
C00470=88.233,-46.990,4.399,-179.9887,0.8564,-928.0383
C00471=86.848,-49.428,4.399,-179.9706,1.7904,-929.6456
C00472=85.672,-51.352,4.398,-179.9249,2.9520,-930.9386
C00473=84.692,-52.853,4.396,-179.8607,4.3050,-931.9667
C00474=83.700,-54.314,4.393,-179.8530,5.6572,-932.9801
C00475=82.455,-56.108,4.390,-179.8953,6.8088,-934.2340
C00476=80.608,-58.679,4.388,-179.9571,7.5869,-936.0529
C00477=77.804,-62.331,4.387,-179.9919,7.8870,-938.6992
C00478=74.450,-66.299,4.387,179.9976,7.9022,-941.6856
C00479=70.493,-70.493,4.387,180.0000,7.9010,-945.0000
C00480=66.299,-74.450,4.387,-179.9976,7.9022,-948.3144
C00481=62.331,-77.804,4.387,179.9919,7.8870,-951.3008
C00482=58.679,-80.608,4.388,179.9571,7.5869,-953.9471
C00483=56.108,-82.455,4.390,179.8953,6.8088,-955.7660
C00484=54.314,-83.700,4.393,179.8530,5.6572,-957.0199
C00485=52.853,-84.692,4.396,179.8607,4.3050,-958.0333
C00486=51.352,-85.672,4.398,179.9249,2.9520,-959.0614
C00487=49.428,-86.848,4.399,179.9706,1.7904,-960.3544
C00488=46.990,-88.233,4.399,179.9887,0.8564,-961.9617
C00489=44.332,-89.625,4.399,179.9990,0.2434,-963.6812
C00490=41.782,-90.851,4.400,179.9987,0.0384,-965.3025
C00491=39.424,-91.901,4.400,-179.9977,0.0053,-966.7815
C00492=37.107,-92.860,4.400,-179.9979,0.0053,-968.2183
C00493=34.697,-93.786,4.400,-179.9988,0.0362,-969.6976
C00494=32.027,-94.722,4.399,-179.9972,0.2410,-971.3188
C00495=29.164,-95.617,4.399,-179.9911,0.8539,-973.0378
C00496=26.460,-96.362,4.399,-179.9728,1.7872,-974.6456
C00497=24.268,-96.890,4.398,-179.9222,2.9528,-975.9384
C00498=22.514,-97.259,4.396,-179.8623,4.3065,-976.9665
C00499=20.779,-97.591,4.393,-179.8518,5.6544,-977.9801
C00500=18.630,-97.979,4.390,-179.8975,6.8083,-979.2341
C00501=15.506,-98.490,4.388,-179.9574,7.5851,-981.0529
C00502=10.941,-99.090,4.387,-179.9908,7.8868,-983.6992
C00503=5.764,-99.524,4.387,179.9969,7.8994,-986.6854
C00504=0.000,-99.691,4.387,180.0000,7.8975,-990.0000
C00505=0.000,-99.691,4.387,180.0000,7.8975,-990.0000
C00506=-5.764,-99.524,4.387,-179.9969,7.8994,-993.3146
C00507=-10.941,-99.090,4.387,179.9908,7.8868,-996.3008
C00508=-15.506,-98.490,4.388,179.9574,7.5851,-998.9471
C00509=-18.630,-97.979,4.390,179.8975,6.8083,-1000.7659
C00510=-20.779,-97.591,4.393,179.8518,5.6544,-1002.0199
C00511=-22.514,-97.259,4.396,179.8623,4.3065,-1003.0335
C00512=-24.268,-96.890,4.398,179.9222,2.9528,-1004.0616
C00513=-26.460,-96.362,4.399,179.9728,1.7872,-1005.3544
C00514=-29.164,-95.617,4.399,179.9911,0.8539,-1006.9622
C00515=-32.027,-94.722,4.399,179.9972,0.2410,-1008.6812
C00516=-34.697,-93.786,4.400,179.9988,0.0362,-1010.3024
C00517=-37.107,-92.860,4.400,179.9979,0.0053,-1011.7817
C00518=-39.424,-91.901,4.400,179.9977,0.0053,-1013.2185
C00519=-41.782,-90.851,4.400,-179.9987,0.0384,-1014.6975
C00520=-44.332,-89.625,4.399,-179.9990,0.2434,-1016.3188
C00521=-46.990,-88.233,4.399,-179.9887,0.8564,-1018.0383
C00522=-49.428,-86.848,4.399,-179.9706,1.7904,-1019.6456
C00523=-51.352,-85.672,4.398,-179.9249,2.9520,-1020.9386
C00524=-52.853,-84.692,4.396,-179.8607,4.3050,-1021.9667
C00525=-54.314,-83.700,4.393,-179.8530,5.6572,-1022.9801
C00526=-56.108,-82.455,4.390,-179.8953,6.8088,-1024.2340
C00527=-58.679,-80.608,4.388,-179.9571,7.5869,-1026.0529
C00528=-62.331,-77.804,4.387,-179.9919,7.8870,-1028.6992
C00529=-66.299,-74.450,4.387,179.9976,7.9022,-1031.6856
C00530=-70.493,-70.493,4.387,-180.0000,7.9010,-1035.0000
C00531=-74.450,-66.299,4.387,-179.9976,7.9022,-1038.3144
C00532=-77.804,-62.331,4.387,179.9919,7.8870,-1041.3008
C00533=-80.608,-58.679,4.388,179.9571,7.5869,-1043.9471
C00534=-82.455,-56.108,4.390,179.8953,6.8088,-1045.7660
C00535=-83.700,-54.314,4.393,179.8530,5.6572,-1047.0199
C00536=-84.692,-52.853,4.396,179.8607,4.3050,-1048.0333
C00537=-85.672,-51.352,4.398,179.9249,2.9520,-1049.0614
C00538=-86.848,-49.428,4.399,179.9706,1.7904,-1050.3544
C00539=-88.233,-46.990,4.399,179.9887,0.8564,-1051.9617
C00540=-89.625,-44.332,4.399,179.9990,0.2434,-1053.6812
C00541=-90.851,-41.782,4.400,179.9987,0.0384,-1055.3025
C00542=-91.901,-39.424,4.400,-179.9977,0.0053,-1056.7815
C00543=-92.860,-37.107,4.400,-179.9979,0.0053,-1058.2183
C00544=-93.786,-34.697,4.400,-179.9988,0.0362,-1059.6976
C00545=-94.722,-32.027,4.399,-179.9972,0.2410,-1061.3188
C00546=-95.617,-29.164,4.399,-179.9911,0.8539,-1063.0378
C00547=-96.362,-26.460,4.399,-179.9728,1.7872,-1064.6456
C00548=-96.890,-24.268,4.398,-179.9222,2.9528,-1065.9384
C00549=-97.259,-22.514,4.396,-179.8623,4.3065,-1066.9665
C00550=-97.591,-20.779,4.393,-179.8518,5.6544,-1067.9801
C00551=-97.979,-18.630,4.390,-179.8975,6.8083,-1069.2341
C00552=-98.490,-15.506,4.388,-179.9574,7.5851,-1071.0529
C00553=-99.090,-10.941,4.387,-179.9908,7.8868,-1073.6992
C00554=-99.524,-5.764,4.387,179.9969,7.8994,-1076.6854
C00555=-99.691,0.000,4.387,-180.0000,7.8975,-1080.0000
C00556=-99.524,5.764,4.387,-179.9969,7.8994,-1083.3146
C00557=-99.090,10.941,4.387,179.9908,7.8868,-1086.3008
C00558=-98.490,15.506,4.388,179.9574,7.5851,-1088.9471
C00559=-97.979,18.630,4.390,179.8975,6.8083,-1090.7659
C00560=-97.591,20.779,4.393,179.8518,5.6544,-1092.0199
C00561=-97.259,22.514,4.396,179.8623,4.3065,-1093.0335
C00562=-96.890,24.268,4.398,179.9222,2.9528,-1094.0616
C00563=-96.362,26.460,4.399,179.9728,1.7872,-1095.3544
C00564=-95.617,29.164,4.399,179.9911,0.8539,-1096.9622
C00565=-94.722,32.027,4.399,179.9972,0.2410,-1098.6812
C00566=-93.786,34.697,4.400,179.9988,0.0362,-1100.3024
C00567=-92.860,37.107,4.400,179.9979,0.0053,-1101.7817
C00568=-91.901,39.424,4.400,179.9977,0.0053,-1103.2185
C00569=-90.851,41.782,4.400,-179.9987,0.0384,-1104.6975
C00570=-89.625,44.332,4.399,-179.9990,0.2434,-1106.3188
C00571=-88.233,46.990,4.399,-179.9887,0.8564,-1108.0383
C00572=-86.848,49.428,4.399,-179.9706,1.7904,-1109.6456
C00573=-85.672,51.352,4.398,-179.9249,2.9520,-1110.9386
C00574=-84.692,52.853,4.396,-179.8607,4.3050,-1111.9667
C00575=-83.700,54.314,4.393,-179.8530,5.6572,-1112.9801
C00576=-82.455,56.108,4.390,-179.8953,6.8088,-1114.2340
C00577=-80.608,58.679,4.388,-179.9571,7.5869,-1116.0529
C00578=-77.804,62.331,4.387,-179.9919,7.8870,-1118.6992
C00579=-74.450,66.299,4.387,179.9976,7.9022,-1121.6856
C00580=-70.493,70.493,4.387,180.0000,7.9010,-1125.0000
C00581=-66.299,74.450,4.387,-179.9976,7.9022,-1128.3144
C00582=-62.331,77.804,4.387,179.9919,7.8870,-1131.3008
C00583=-58.679,80.608,4.388,179.9571,7.5869,-1133.9471
C00584=-56.108,82.455,4.390,179.8953,6.8088,-1135.7660
C00585=-54.314,83.700,4.393,179.8530,5.6572,-1137.0199
C00586=-52.853,84.692,4.396,179.8607,4.3050,-1138.0333
C00587=-51.352,85.672,4.398,179.9249,2.9520,-1139.0614
C00588=-49.428,86.848,4.399,179.9706,1.7904,-1140.3544
C00589=-46.990,88.233,4.399,179.9887,0.8564,-1141.9617
C00590=-44.332,89.625,4.399,179.9990,0.2434,-1143.6812
C00591=-41.782,90.851,4.400,179.9987,0.0384,-1145.3025
C00592=-39.424,91.901,4.400,-179.9977,0.0053,-1146.7815
C00593=-37.107,92.860,4.400,-179.9979,0.0053,-1148.2183
C00594=-34.697,93.786,4.400,-179.9988,0.0362,-1149.6976
C00595=-32.027,94.722,4.399,-179.9972,0.2410,-1151.3188
C00596=-29.164,95.617,4.399,-179.9911,0.8539,-1153.0378
C00597=-26.460,96.362,4.399,-179.9728,1.7872,-1154.6456
C00598=-24.268,96.890,4.398,-179.9222,2.9528,-1155.9384
C00599=-22.514,97.259,4.396,-179.8623,4.3065,-1156.9665
C00600=-20.779,97.591,4.393,-179.8518,5.6544,-1157.9801
C00601=-18.630,97.979,4.390,-179.8975,6.8083,-1159.2341
C00602=-15.506,98.490,4.388,-179.9574,7.5851,-1161.0529
C00603=-10.941,99.090,4.387,-179.9908,7.8868,-1163.6992
C00604=-5.764,99.524,4.387,179.9969,7.8994,-1166.6854
C00605=0.000,99.691,4.387,180.0000,7.8975,-1170.0000
C00606=0.000,99.321,6.555,180.0000,11.4729,-1170.0000
C00607=5.730,99.155,6.555,-179.9986,11.4747,-1173.3073
C00608=10.884,98.723,6.555,179.9789,11.4524,-1176.2913
C00609=15.437,98.140,6.558,179.8697,11.0220,-1178.9391
C00610=18.547,97.668,6.566,179.6614,9.8830,-1180.7524
C00611=20.687,97.336,6.576,179.5149,8.1850,-1181.9986
C00612=22.417,97.071,6.585,179.5571,6.1969,-1183.0036
C00613=24.167,96.770,6.592,179.7516,4.2352,-1184.0220
C00614=26.351,96.303,6.595,179.9073,2.5536,-1185.3030
C00615=29.062,95.605,6.597,179.9725,1.2134,-1186.9082
C00616=31.947,94.737,6.598,179.9952,0.3370,-1188.6350
C00617=34.646,93.803,6.599,179.9983,0.0543,-1190.2716
C00618=37.090,92.867,6.600,179.9979,0.0053,-1191.7712
C00619=39.440,91.893,6.600,179.9977,0.0053,-1193.2288
C00620=41.830,90.827,6.599,179.9992,0.0564,-1194.7282
C00621=44.399,89.579,6.598,-179.9937,0.3356,-1196.3649
C00622=47.053,88.152,6.597,-179.9707,1.2107,-1198.0920
C00623=49.464,86.729,6.595,-179.9090,2.5592,-1199.6973
C00624=51.338,85.515,6.592,-179.7528,4.2349,-1200.9780
C00625=52.788,84.491,6.585,-179.5585,6.1980,-1201.9962
C00626=54.199,83.455,6.576,-179.5155,8.1891,-1203.0013
C00627=55.947,82.176,6.566,-179.6616,9.8834,-1204.2478
C00628=58.480,80.311,6.558,-179.8658,11.0226,-1206.0610
C00629=62.112,77.504,6.555,-179.9807,11.4500,-1208.7088
C00630=66.061,74.165,6.555,179.9973,11.4763,-1211.6924
C00631=70.230,70.230,6.555,-180.0000,11.4694,-1215.0000
C00632=74.165,66.061,6.555,-179.9973,11.4763,-1218.3076
C00633=77.504,62.112,6.555,179.9807,11.4500,-1221.2912
C00634=80.311,58.480,6.558,179.8658,11.0226,-1223.9390
C00635=82.176,55.947,6.566,179.6616,9.8834,-1225.7522
C00636=83.455,54.199,6.576,179.5155,8.1891,-1226.9987
C00637=84.491,52.788,6.585,179.5585,6.1980,-1228.0038
C00638=85.515,51.338,6.592,179.7528,4.2349,-1229.0220
C00639=86.729,49.464,6.595,179.9090,2.5592,-1230.3027
C00640=88.152,47.053,6.597,179.9707,1.2107,-1231.9080
C00641=89.579,44.399,6.598,179.9937,0.3356,-1233.6351
C00642=90.827,41.830,6.599,-179.9992,0.0564,-1235.2718
C00643=91.893,39.440,6.600,-179.9977,0.0053,-1236.7712
C00644=92.867,37.090,6.600,-179.9979,0.0053,-1238.2288
C00645=93.803,34.646,6.599,-179.9983,0.0543,-1239.7284
C00646=94.737,31.947,6.598,-179.9952,0.3370,-1241.3650
C00647=95.605,29.062,6.597,-179.9725,1.2134,-1243.0918
C00648=96.303,26.351,6.595,-179.9073,2.5536,-1244.6970
C00649=96.770,24.167,6.592,-179.7516,4.2352,-1245.9780
C00650=97.071,22.417,6.585,-179.5571,6.1969,-1246.9964
C00651=97.336,20.687,6.576,-179.5149,8.1850,-1248.0014
C00652=97.668,18.547,6.566,-179.6614,9.8830,-1249.2476
C00653=98.140,15.437,6.558,-179.8697,11.0220,-1251.0609
C00654=98.723,10.884,6.555,-179.9789,11.4524,-1253.7087
C00655=99.155,5.730,6.555,179.9986,11.4747,-1256.6927
C00656=99.321,0.000,6.555,-180.0000,11.4729,-1260.0000
C00657=99.155,-5.730,6.555,-179.9986,11.4747,-1263.3073
C00658=98.723,-10.884,6.555,179.9789,11.4524,-1266.2913
C00659=98.140,-15.437,6.558,179.8697,11.0220,-1268.9391
C00660=97.668,-18.547,6.566,179.6614,9.8830,-1270.7524
C00661=97.336,-20.687,6.576,179.5149,8.1850,-1271.9986
C00662=97.071,-22.417,6.585,179.5571,6.1969,-1273.0036
C00663=96.770,-24.167,6.592,179.7516,4.2352,-1274.0220
C00664=96.303,-26.351,6.595,179.9073,2.5536,-1275.3030
C00665=95.605,-29.062,6.597,179.9725,1.2134,-1276.9082
C00666=94.737,-31.947,6.598,179.9952,0.3370,-1278.6350
C00667=93.803,-34.646,6.599,179.9983,0.0543,-1280.2716
C00668=92.867,-37.090,6.600,179.9979,0.0053,-1281.7712
C00669=91.893,-39.440,6.600,179.9977,0.0053,-1283.2288
C00670=90.827,-41.830,6.599,179.9992,0.0564,-1284.7282
C00671=89.579,-44.399,6.598,-179.9937,0.3356,-1286.3649
C00672=88.152,-47.053,6.597,-179.9707,1.2107,-1288.0920
C00673=86.729,-49.464,6.595,-179.9090,2.5592,-1289.6973
C00674=85.515,-51.338,6.592,-179.7528,4.2349,-1290.9780
C00675=84.491,-52.788,6.585,-179.5585,6.1980,-1291.9962
C00676=83.455,-54.199,6.576,-179.5155,8.1891,-1293.0013
C00677=82.176,-55.947,6.566,-179.6616,9.8834,-1294.2478
C00678=80.311,-58.480,6.558,-179.8658,11.0226,-1296.0610
C00679=77.504,-62.112,6.555,-179.9807,11.4500,-1298.7088
C00680=74.165,-66.061,6.555,179.9973,11.4763,-1301.6924
C00681=70.230,-70.230,6.555,-180.0000,11.4694,-1305.0000
C00682=66.061,-74.165,6.555,-179.9973,11.4763,-1308.3076
C00683=62.112,-77.504,6.555,179.9807,11.4500,-1311.2912
C00684=58.480,-80.311,6.558,179.8658,11.0226,-1313.9390
C00685=55.947,-82.176,6.566,179.6616,9.8834,-1315.7522
C00686=54.199,-83.455,6.576,179.5155,8.1891,-1316.9987
C00687=52.788,-84.491,6.585,179.5585,6.1980,-1318.0038
C00688=51.338,-85.515,6.592,179.7528,4.2349,-1319.0220
C00689=49.464,-86.729,6.595,179.9090,2.5592,-1320.3027
C00690=47.053,-88.152,6.597,179.9707,1.2107,-1321.9080
C00691=44.399,-89.579,6.598,179.9937,0.3356,-1323.6351
C00692=41.830,-90.827,6.599,-179.9992,0.0564,-1325.2718
C00693=39.440,-91.893,6.600,-179.9977,0.0053,-1326.7712
C00694=37.090,-92.867,6.600,-179.9979,0.0053,-1328.2288
C00695=34.646,-93.803,6.599,-179.9983,0.0543,-1329.7284
C00696=31.947,-94.737,6.598,-179.9952,0.3370,-1331.3650
C00697=29.062,-95.605,6.597,-179.9725,1.2134,-1333.0918
C00698=26.351,-96.303,6.595,-179.9073,2.5536,-1334.6970
C00699=24.167,-96.770,6.592,-179.7516,4.2352,-1335.9780
C00700=22.417,-97.071,6.585,-179.5571,6.1969,-1336.9964
C00701=20.687,-97.336,6.576,-179.5149,8.1850,-1338.0014
C00702=18.547,-97.668,6.566,-179.6614,9.8830,-1339.2476
C00703=15.437,-98.140,6.558,-179.8697,11.0220,-1341.0609
C00704=10.884,-98.723,6.555,-179.9789,11.4524,-1343.7087
C00705=5.730,-99.155,6.555,179.9986,11.4747,-1346.6927
C00706=0.000,-99.321,6.555,180.0000,11.4729,-1350.0000
C00707=0.000,-99.321,6.555,180.0000,11.4729,-1350.0000
C00708=-5.730,-99.155,6.555,-179.9986,11.4747,-1353.3073
C00709=-10.884,-98.723,6.555,179.9789,11.4524,-1356.2913
C00710=-15.437,-98.140,6.558,179.8697,11.0220,-1358.9391
C00711=-18.547,-97.668,6.566,179.6614,9.8830,-1360.7524
C00712=-20.687,-97.336,6.576,179.5149,8.1850,-1361.9986
C00713=-22.417,-97.071,6.585,179.5571,6.1969,-1363.0036
C00714=-24.167,-96.770,6.592,179.7516,4.2352,-1364.0220
C00715=-26.351,-96.303,6.595,179.9073,2.5536,-1365.3030
C00716=-29.062,-95.605,6.597,179.9725,1.2134,-1366.9082
C00717=-31.947,-94.737,6.598,179.9952,0.3370,-1368.6350
C00718=-34.646,-93.803,6.599,179.9983,0.0543,-1370.2716
C00719=-37.090,-92.867,6.600,179.9979,0.0053,-1371.7712
C00720=-39.440,-91.893,6.600,179.9977,0.0053,-1373.2288
C00721=-41.830,-90.827,6.599,179.9992,0.0564,-1374.7282
C00722=-44.399,-89.579,6.598,-179.9937,0.3356,-1376.3649
C00723=-47.053,-88.152,6.597,-179.9707,1.2107,-1378.0920
C00724=-49.464,-86.729,6.595,-179.9090,2.5592,-1379.6973
C00725=-51.338,-85.515,6.592,-179.7528,4.2349,-1380.9780
C00726=-52.788,-84.491,6.585,-179.5585,6.1980,-1381.9962
C00727=-54.199,-83.455,6.576,-179.5155,8.1891,-1383.0013
C00728=-55.947,-82.176,6.566,-179.6616,9.8834,-1384.2478
C00729=-58.480,-80.311,6.558,-179.8658,11.0226,-1386.0610
C00730=-62.112,-77.504,6.555,-179.9807,11.4500,-1388.7088
C00731=-66.061,-74.165,6.555,179.9973,11.4763,-1391.6924
C00732=-70.230,-70.230,6.555,-180.0000,11.4694,-1395.0000
C00733=-74.165,-66.061,6.555,-179.9973,11.4763,-1398.3076
C00734=-77.504,-62.112,6.555,179.9807,11.4500,-1401.2912
C00735=-80.311,-58.480,6.558,179.8658,11.0226,-1403.9390
C00736=-82.176,-55.947,6.566,179.6616,9.8834,-1405.7522
C00737=-83.455,-54.199,6.576,179.5155,8.1891,-1406.9987
C00738=-84.491,-52.788,6.585,179.5585,6.1980,-1408.0038
C00739=-85.515,-51.338,6.592,179.7528,4.2349,-1409.0220
C00740=-86.729,-49.464,6.595,179.9090,2.5592,-1410.3027
C00741=-88.152,-47.053,6.597,179.9707,1.2107,-1411.9080
C00742=-89.579,-44.399,6.598,179.9937,0.3356,-1413.6351
C00743=-90.827,-41.830,6.599,-179.9992,0.0564,-1415.2718
C00744=-91.893,-39.440,6.600,-179.9977,0.0053,-1416.7712
C00745=-92.867,-37.090,6.600,-179.9979,0.0053,-1418.2288
C00746=-93.803,-34.646,6.599,-179.9983,0.0543,-1419.7284
C00747=-94.737,-31.947,6.598,-179.9952,0.3370,-1421.3650
C00748=-95.605,-29.062,6.597,-179.9725,1.2134,-1423.0918
C00749=-96.303,-26.351,6.595,-179.9073,2.5536,-1424.6970
C00750=-96.770,-24.167,6.592,-179.7516,4.2352,-1425.9780
C00751=-97.071,-22.417,6.585,-179.5571,6.1969,-1426.9964
C00752=-97.336,-20.687,6.576,-179.5149,8.1850,-1428.0014
C00753=-97.668,-18.547,6.566,-179.6614,9.8830,-1429.2476
C00754=-98.140,-15.437,6.558,-179.8697,11.0220,-1431.0609
C00755=-98.723,-10.884,6.555,-179.9789,11.4524,-1433.7087
C00756=-99.155,-5.730,6.555,179.9986,11.4747,-1436.6927
C00757=-99.321,0.000,6.555,-180.0000,11.4729,-1440.0000
C00758=-99.155,5.730,6.555,-179.9986,11.4747,-1443.3073
C00759=-98.723,10.884,6.555,179.9789,11.4524,-1446.2913
C00760=-98.140,15.437,6.558,179.8697,11.0220,-1448.9391
C00761=-97.668,18.547,6.566,179.6614,9.8830,-1450.7524
C00762=-97.336,20.687,6.576,179.5149,8.1850,-1451.9986
C00763=-97.071,22.417,6.585,179.5571,6.1969,-1453.0036
C00764=-96.770,24.167,6.592,179.7516,4.2352,-1454.0220
C00765=-96.303,26.351,6.595,179.9073,2.5536,-1455.3030
C00766=-95.605,29.062,6.597,179.9725,1.2134,-1456.9082
C00767=-94.737,31.947,6.598,179.9952,0.3370,-1458.6350
C00768=-93.803,34.646,6.599,179.9983,0.0543,-1460.2716
C00769=-92.867,37.090,6.600,179.9979,0.0053,-1461.7712
C00770=-91.893,39.440,6.600,179.9977,0.0053,-1463.2288
C00771=-90.827,41.830,6.599,179.9992,0.0564,-1464.7282
C00772=-89.579,44.399,6.598,-179.9937,0.3356,-1466.3649
C00773=-88.152,47.053,6.597,-179.9707,1.2107,-1468.0920
C00774=-86.729,49.464,6.595,-179.9090,2.5592,-1469.6973
C00775=-85.515,51.338,6.592,-179.7528,4.2349,-1470.9780
C00776=-84.491,52.788,6.585,-179.5585,6.1980,-1471.9962
C00777=-83.455,54.199,6.576,-179.5155,8.1891,-1473.0013
C00778=-82.176,55.947,6.566,-179.6616,9.8834,-1474.2478
C00779=-80.311,58.480,6.558,-179.8658,11.0226,-1476.0610
C00780=-77.504,62.112,6.555,-179.9807,11.4500,-1478.7088
C00781=-74.165,66.061,6.555,179.9973,11.4763,-1481.6924
C00782=-70.230,70.230,6.555,-180.0000,11.4694,-1485.0000
C00783=-66.061,74.165,6.555,-179.9973,11.4763,-1488.3076
C00784=-62.112,77.504,6.555,179.9807,11.4500,-1491.2912
C00785=-58.480,80.311,6.558,179.8658,11.0226,-1493.9390
C00786=-55.947,82.176,6.566,179.6616,9.8834,-1495.7522
C00787=-54.199,83.455,6.576,179.5155,8.1891,-1496.9987
C00788=-52.788,84.491,6.585,179.5585,6.1980,-1498.0038
C00789=-51.338,85.515,6.592,179.7528,4.2349,-1499.0220
C00790=-49.464,86.729,6.595,179.9090,2.5592,-1500.3027
C00791=-47.053,88.152,6.597,179.9707,1.2107,-1501.9080
C00792=-44.399,89.579,6.598,179.9937,0.3356,-1503.6351
C00793=-41.830,90.827,6.599,-179.9992,0.0564,-1505.2718
C00794=-39.440,91.893,6.600,-179.9977,0.0053,-1506.7712
C00795=-37.090,92.867,6.600,-179.9979,0.0053,-1508.2288
C00796=-34.646,93.803,6.599,-179.9983,0.0543,-1509.7284
C00797=-31.947,94.737,6.598,-179.9952,0.3370,-1511.3650
C00798=-29.062,95.605,6.597,-179.9725,1.2134,-1513.0918
C00799=-26.351,96.303,6.595,-179.9073,2.5536,-1514.6970
C00800=-24.167,96.770,6.592,-179.7516,4.2352,-1515.9780
C00801=-22.417,97.071,6.585,-179.5571,6.1969,-1516.9964
C00802=-20.687,97.336,6.576,-179.5149,8.1850,-1518.0014
C00803=-18.547,97.668,6.566,-179.6614,9.8830,-1519.2476
C00804=-15.437,98.140,6.558,-179.8697,11.0220,-1521.0609
C00805=-10.884,98.723,6.555,-179.9789,11.4524,-1523.7087
C00806=-5.730,99.155,6.555,179.9986,11.4747,-1526.6927
C00807=0.000,99.321,6.555,180.0000,11.4729,-1530.0000
C00808=0.000,98.820,8.697,180.0000,14.7616,-1530.0000
C00809=5.684,98.656,8.697,-179.9919,14.7688,-1533.2974
C00810=10.807,98.229,8.698,179.9574,14.7351,-1536.2783
C00811=15.344,97.668,8.705,179.6987,14.1865,-1538.9284
C00812=18.436,97.247,8.723,179.2265,12.6975,-1540.7347
C00813=20.563,96.991,8.745,178.9035,10.4501,-1541.9700
C00814=22.286,96.814,8.767,179.0085,7.8426,-1542.9633
C00815=24.029,96.606,8.782,179.4467,5.3324,-1543.9678
C00816=26.202,96.222,8.789,179.7964,3.2124,-1545.2327
C00817=28.922,95.588,8.792,179.9388,1.5081,-1546.8342
C00818=31.837,94.757,8.795,179.9918,0.4022,-1548.5716
C00819=34.577,93.826,8.798,179.9997,0.0671,-1550.2300
C00820=37.066,92.876,8.800,-179.9968,0.0074,-1551.7565
C00821=39.463,91.883,8.800,-179.9970,0.0075,-1553.2431
C00822=41.895,90.794,8.798,179.9996,0.0692,-1554.7700
C00823=44.491,89.515,8.795,-179.9888,0.4023,-1556.4284
C00824=47.140,88.042,8.792,-179.9421,1.5064,-1558.1658
C00825=49.511,86.567,8.789,-179.7969,3.2134,-1559.7669
C00826=51.320,85.302,8.782,-179.4498,5.3325,-1561.0323
C00827=52.699,84.217,8.767,-179.0068,7.8395,-1562.0364
C00828=54.043,83.124,8.745,-178.9053,10.4506,-1563.0299
C00829=55.728,81.800,8.723,-179.2272,12.6950,-1564.2655
C00830=58.212,79.911,8.705,-179.7001,14.1862,-1566.0719
C00831=61.817,77.101,8.698,-179.9561,14.7367,-1568.7215
C00832=65.741,73.780,8.697,179.9932,14.7681,-1571.7023
C00833=69.877,69.877,8.697,-180.0000,14.7639,-1575.0000
C00834=73.780,65.741,8.697,-179.9932,14.7681,-1578.2977
C00835=77.101,61.817,8.698,179.9561,14.7367,-1581.2785
C00836=79.911,58.212,8.705,179.7001,14.1862,-1583.9281
C00837=81.800,55.728,8.723,179.2272,12.6950,-1585.7345
C00838=83.124,54.043,8.745,178.9053,10.4506,-1586.9701
C00839=84.217,52.699,8.767,179.0068,7.8395,-1587.9636
C00840=85.302,51.320,8.782,179.4498,5.3325,-1588.9677
C00841=86.567,49.511,8.789,179.7969,3.2134,-1590.2331
C00842=88.042,47.140,8.792,179.9421,1.5064,-1591.8342
C00843=89.515,44.491,8.795,179.9888,0.4023,-1593.5716
C00844=90.794,41.895,8.798,-179.9996,0.0692,-1595.2300
C00845=91.883,39.463,8.800,179.9970,0.0075,-1596.7569
C00846=92.876,37.066,8.800,179.9968,0.0074,-1598.2435
C00847=93.826,34.577,8.798,-179.9997,0.0671,-1599.7700
C00848=94.757,31.837,8.795,-179.9918,0.4022,-1601.4284
C00849=95.588,28.922,8.792,-179.9388,1.5081,-1603.1658
C00850=96.222,26.202,8.789,-179.7964,3.2124,-1604.7673
C00851=96.606,24.029,8.782,-179.4467,5.3324,-1606.0322
C00852=96.814,22.286,8.767,-179.0085,7.8426,-1607.0367
C00853=96.991,20.563,8.745,-178.9035,10.4501,-1608.0300
C00854=97.247,18.436,8.723,-179.2265,12.6975,-1609.2653
C00855=97.668,15.344,8.705,-179.6987,14.1865,-1611.0716
C00856=98.229,10.807,8.698,-179.9574,14.7351,-1613.7217
C00857=98.656,5.684,8.697,179.9919,14.7688,-1616.7026
C00858=98.820,0.000,8.697,-180.0000,14.7616,-1620.0000
C00859=98.656,-5.684,8.697,-179.9919,14.7688,-1623.2974
C00860=98.229,-10.807,8.698,179.9574,14.7351,-1626.2783
C00861=97.668,-15.344,8.705,179.6987,14.1865,-1628.9284
C00862=97.247,-18.436,8.723,179.2265,12.6975,-1630.7347
C00863=96.991,-20.563,8.745,178.9035,10.4501,-1631.9700
C00864=96.814,-22.286,8.767,179.0085,7.8426,-1632.9633
C00865=96.606,-24.029,8.782,179.4467,5.3324,-1633.9678
C00866=96.222,-26.202,8.789,179.7964,3.2124,-1635.2327
C00867=95.588,-28.922,8.792,179.9388,1.5081,-1636.8342
C00868=94.757,-31.837,8.795,179.9918,0.4022,-1638.5716
C00869=93.826,-34.577,8.798,179.9997,0.0671,-1640.2300
C00870=92.876,-37.066,8.800,-179.9968,0.0074,-1641.7565
C00871=91.883,-39.463,8.800,-179.9970,0.0075,-1643.2431
C00872=90.794,-41.895,8.798,179.9996,0.0692,-1644.7700
C00873=89.515,-44.491,8.795,-179.9888,0.4023,-1646.4284
C00874=88.042,-47.140,8.792,-179.9421,1.5064,-1648.1658
C00875=86.567,-49.511,8.789,-179.7969,3.2134,-1649.7669
C00876=85.302,-51.320,8.782,-179.4498,5.3325,-1651.0323
C00877=84.217,-52.699,8.767,-179.0068,7.8395,-1652.0364
C00878=83.124,-54.043,8.745,-178.9053,10.4506,-1653.0299
C00879=81.800,-55.728,8.723,-179.2272,12.6950,-1654.2655
C00880=79.911,-58.212,8.705,-179.7001,14.1862,-1656.0719
C00881=77.101,-61.817,8.698,-179.9561,14.7367,-1658.7215
C00882=73.780,-65.741,8.697,179.9932,14.7681,-1661.7023
C00883=69.877,-69.877,8.697,-180.0000,14.7639,-1665.0000
C00884=65.741,-73.780,8.697,-179.9932,14.7681,-1668.2977
C00885=61.817,-77.101,8.698,179.9561,14.7367,-1671.2785
C00886=58.212,-79.911,8.705,179.7001,14.1862,-1673.9281
C00887=55.728,-81.800,8.723,179.2272,12.6950,-1675.7345
C00888=54.043,-83.124,8.745,178.9053,10.4506,-1676.9701
C00889=52.699,-84.217,8.767,179.0068,7.8395,-1677.9636
C00890=51.320,-85.302,8.782,179.4498,5.3325,-1678.9677
C00891=49.511,-86.567,8.789,179.7969,3.2134,-1680.2331
C00892=47.140,-88.042,8.792,179.9421,1.5064,-1681.8342
C00893=44.491,-89.515,8.795,179.9888,0.4023,-1683.5716
C00894=41.895,-90.794,8.798,-179.9996,0.0692,-1685.2300
C00895=39.463,-91.883,8.800,179.9970,0.0075,-1686.7569
C00896=37.066,-92.876,8.800,179.9968,0.0074,-1688.2435
C00897=34.577,-93.826,8.798,-179.9997,0.0671,-1689.7700
C00898=31.837,-94.757,8.795,-179.9918,0.4022,-1691.4284
C00899=28.922,-95.588,8.792,-179.9388,1.5081,-1693.1658
C00900=26.202,-96.222,8.789,-179.7964,3.2124,-1694.7673
C00901=24.029,-96.606,8.782,-179.4467,5.3324,-1696.0322
C00902=22.286,-96.814,8.767,-179.0085,7.8426,-1697.0367
C00903=20.563,-96.991,8.745,-178.9035,10.4501,-1698.0300
C00904=18.436,-97.247,8.723,-179.2265,12.6975,-1699.2653
C00905=15.344,-97.668,8.705,-179.6987,14.1865,-1701.0716
C00906=10.807,-98.229,8.698,-179.9574,14.7351,-1703.7217
C00907=5.684,-98.656,8.697,179.9919,14.7688,-1706.7026
C00908=0.000,-98.820,8.697,180.0000,14.7616,-1710.0000
C00909=0.000,-98.820,8.697,180.0000,14.7616,-1710.0000
C00910=-5.684,-98.656,8.697,-179.9919,14.7688,-1713.2974
C00911=-10.807,-98.229,8.698,179.9574,14.7351,-1716.2783
C00912=-15.344,-97.668,8.705,179.6987,14.1865,-1718.9284
C00913=-18.436,-97.247,8.723,179.2265,12.6975,-1720.7347
C00914=-20.563,-96.991,8.745,178.9035,10.4501,-1721.9700
C00915=-22.286,-96.814,8.767,179.0085,7.8426,-1722.9633
C00916=-24.029,-96.606,8.782,179.4467,5.3324,-1723.9678
C00917=-26.202,-96.222,8.789,179.7964,3.2124,-1725.2327
C00918=-28.922,-95.588,8.792,179.9388,1.5081,-1726.8342
C00919=-31.837,-94.757,8.795,179.9918,0.4022,-1728.5716
C00920=-34.577,-93.826,8.798,179.9997,0.0671,-1730.2300
C00921=-37.066,-92.876,8.800,-179.9968,0.0074,-1731.7565
C00922=-39.463,-91.883,8.800,-179.9970,0.0075,-1733.2431
C00923=-41.895,-90.794,8.798,179.9996,0.0692,-1734.7700
C00924=-44.491,-89.515,8.795,-179.9888,0.4023,-1736.4284
C00925=-47.140,-88.042,8.792,-179.9421,1.5064,-1738.1658
C00926=-49.511,-86.567,8.789,-179.7969,3.2134,-1739.7669
C00927=-51.320,-85.302,8.782,-179.4498,5.3325,-1741.0323
C00928=-52.699,-84.217,8.767,-179.0068,7.8395,-1742.0364
C00929=-54.043,-83.124,8.745,-178.9053,10.4506,-1743.0299
C00930=-55.728,-81.800,8.723,-179.2272,12.6950,-1744.2655
C00931=-58.212,-79.911,8.705,-179.7001,14.1862,-1746.0719
C00932=-61.817,-77.101,8.698,-179.9561,14.7367,-1748.7215
C00933=-65.741,-73.780,8.697,179.9932,14.7681,-1751.7023
C00934=-69.877,-69.877,8.697,-180.0000,14.7639,-1755.0000
C00935=-73.780,-65.741,8.697,-179.9932,14.7681,-1758.2977
C00936=-77.101,-61.817,8.698,179.9561,14.7367,-1761.2785
C00937=-79.911,-58.212,8.705,179.7001,14.1862,-1763.9281
C00938=-81.800,-55.728,8.723,179.2272,12.6950,-1765.7345
C00939=-83.124,-54.043,8.745,178.9053,10.4506,-1766.9701
C00940=-84.217,-52.699,8.767,179.0068,7.8395,-1767.9636
C00941=-85.302,-51.320,8.782,179.4498,5.3325,-1768.9677
C00942=-86.567,-49.511,8.789,179.7969,3.2134,-1770.2331
C00943=-88.042,-47.140,8.792,179.9421,1.5064,-1771.8342
C00944=-89.515,-44.491,8.795,179.9888,0.4023,-1773.5716
C00945=-90.794,-41.895,8.798,-179.9996,0.0692,-1775.2300
C00946=-91.883,-39.463,8.800,179.9970,0.0075,-1776.7569
C00947=-92.876,-37.066,8.800,179.9968,0.0074,-1778.2435
C00948=-93.826,-34.577,8.798,-179.9997,0.0671,-1779.7700
C00949=-94.757,-31.837,8.795,-179.9918,0.4022,-1781.4284
C00950=-95.588,-28.922,8.792,-179.9388,1.5081,-1783.1658
C00951=-96.222,-26.202,8.789,-179.7964,3.2124,-1784.7673
C00952=-96.606,-24.029,8.782,-179.4467,5.3324,-1786.0322
C00953=-96.814,-22.286,8.767,-179.0085,7.8426,-1787.0367
C00954=-96.991,-20.563,8.745,-178.9035,10.4501,-1788.0300
C00955=-97.247,-18.436,8.723,-179.2265,12.6975,-1789.2653
C00956=-97.668,-15.344,8.705,-179.6987,14.1865,-1791.0716
C00957=-98.229,-10.807,8.698,-179.9574,14.7351,-1793.7217
C00958=-98.656,-5.684,8.697,179.9919,14.7688,-1796.7026
C00959=-98.820,0.000,8.697,-180.0000,14.7616,-1800.0000
C00960=-98.656,5.684,8.697,-179.9919,14.7688,-1803.2974
C00961=-98.229,10.807,8.698,179.9574,14.7351,-1806.2783
C00962=-97.668,15.344,8.705,179.6987,14.1865,-1808.9284
C00963=-97.247,18.436,8.723,179.2265,12.6975,-1810.7347
C00964=-96.991,20.563,8.745,178.9035,10.4501,-1811.9700
C00965=-96.814,22.286,8.767,179.0085,7.8426,-1812.9633
C00966=-96.606,24.029,8.782,179.4467,5.3324,-1813.9678
C00967=-96.222,26.202,8.789,179.7964,3.2124,-1815.2327
C00968=-95.588,28.922,8.792,179.9388,1.5081,-1816.8342
C00969=-94.757,31.837,8.795,179.9918,0.4022,-1818.5716
C00970=-93.826,34.577,8.798,179.9997,0.0671,-1820.2300
C00971=-92.876,37.066,8.800,-179.9968,0.0074,-1821.7565
C00972=-91.883,39.463,8.800,-179.9970,0.0075,-1823.2431
C00973=-90.794,41.895,8.798,179.9996,0.0692,-1824.7700
C00974=-89.515,44.491,8.795,-179.9888,0.4023,-1826.4284
C00975=-88.042,47.140,8.792,-179.9421,1.5064,-1828.1658
C00976=-86.567,49.511,8.789,-179.7969,3.2134,-1829.7669
C00977=-85.302,51.320,8.782,-179.4498,5.3325,-1831.0323
C00978=-84.217,52.699,8.767,-179.0068,7.8395,-1832.0364
C00979=-83.124,54.043,8.745,-178.9053,10.4506,-1833.0299
C00980=-81.800,55.728,8.723,-179.2272,12.6950,-1834.2655
C00981=-79.911,58.212,8.705,-179.7001,14.1862,-1836.0719
C00982=-77.101,61.817,8.698,-179.9561,14.7367,-1838.7215
C00983=-73.780,65.741,8.697,179.9932,14.7681,-1841.7023
C00984=-69.877,69.877,8.697,-180.0000,14.7639,-1845.0000
C00985=-65.741,73.780,8.697,-179.9932,14.7681,-1848.2977
C00986=-61.817,77.101,8.698,179.9561,14.7367,-1851.2785
C00987=-58.212,79.911,8.705,179.7001,14.1862,-1853.9281
C00988=-55.728,81.800,8.723,179.2272,12.6950,-1855.7345
C00989=-54.043,83.124,8.745,178.9053,10.4506,-1856.9701
C00990=-52.699,84.217,8.767,179.0068,7.8395,-1857.9636
C00991=-51.320,85.302,8.782,179.4498,5.3325,-1858.9677
C00992=-49.511,86.567,8.789,179.7969,3.2134,-1860.2331
C00993=-47.140,88.042,8.792,179.9421,1.5064,-1861.8342
C00994=-44.491,89.515,8.795,179.9888,0.4023,-1863.5716
C00995=-41.895,90.794,8.798,-179.9996,0.0692,-1865.2300
C00996=-39.463,91.883,8.800,179.9970,0.0075,-1866.7569
C00997=-37.066,92.876,8.800,179.9968,0.0074,-1868.2435
C00998=-34.577,93.826,8.798,-179.9997,0.0671,-1869.7700
C00999=-31.837,94.757,8.795,-179.9918,0.4022,-1871.4284
C01000=-28.922,95.588,8.792,-179.9388,1.5081,-1873.1658
C01001=-26.202,96.222,8.789,-179.7964,3.2124,-1874.7673
C01002=-24.029,96.606,8.782,-179.4467,5.3324,-1876.0322
C01003=-22.286,96.814,8.767,-179.0085,7.8426,-1877.0367
C01004=-20.563,96.991,8.745,-178.9035,10.4501,-1878.0300
C01005=-18.436,97.247,8.723,-179.2265,12.6975,-1879.2653
C01006=-15.344,97.668,8.705,-179.6987,14.1865,-1881.0716
C01007=-10.807,98.229,8.698,-179.9574,14.7351,-1883.7217
C01008=-5.684,98.656,8.697,179.9919,14.7688,-1886.7026
C01009=0.000,98.820,8.697,180.0000,14.7616,-1890.0000
C01010=0.000,98.204,10.809,180.0000,17.7591,-1890.0000
C01011=5.628,98.041,10.809,-179.9935,17.7704,-1893.2854
C01012=10.712,97.620,10.809,179.9140,17.7316,-1896.2621
C01013=15.229,97.084,10.823,179.4369,17.0680,-1898.9150
C01014=18.298,96.727,10.856,178.5506,15.2200,-1900.7121
C01015=20.409,96.562,10.898,177.9749,12.3697,-1901.9342
C01016=22.123,96.495,10.937,178.1855,9.1378,-1902.9128
C01017=23.856,96.400,10.965,178.9958,6.1937,-1903.8997
C01018=26.016,96.121,10.978,179.6325,3.7259,-1905.1448
C01019=28.748,95.567,10.985,179.8949,1.7218,-1906.7421
C01020=31.699,94.782,10.991,179.9869,0.4366,-1908.4921
C01021=34.490,93.854,10.996,-179.9988,0.0798,-1910.1777
C01022=37.037,92.887,11.000,-179.9968,0.0074,-1911.7387
C01023=39.492,91.870,11.000,-179.9970,0.0075,-1913.2613
C01024=41.977,90.753,10.996,-179.9977,0.0768,-1914.8225
C01025=44.606,89.436,10.991,-179.9868,0.4356,-1916.5076
C01026=47.248,87.904,10.985,-179.8919,1.7236,-1918.2578
C01027=49.571,86.364,10.978,-179.6333,3.7272,-1919.8549
C01028=51.296,85.034,10.965,-178.9987,6.1941,-1921.1001
C01029=52.589,83.875,10.937,-178.1865,9.1389,-1922.0874
C01030=53.849,82.711,10.898,-177.9740,12.3647,-1923.0661
C01031=55.458,81.334,10.856,-178.5518,15.2206,-1924.2883
C01032=57.880,79.417,10.823,-179.4413,17.0686,-1926.0850
C01033=61.453,76.603,10.809,-179.9149,17.7331,-1928.7375
C01034=65.346,73.305,10.809,179.9930,17.7700,-1931.7146
C01035=69.440,69.440,10.809,-180.0000,17.7616,-1935.0000
C01036=73.305,65.346,10.809,-179.9930,17.7700,-1938.2854
C01037=76.603,61.453,10.809,179.9149,17.7331,-1941.2625
C01038=79.417,57.880,10.823,179.4413,17.0686,-1943.9150
C01039=81.334,55.458,10.856,178.5518,15.2206,-1945.7117
C01040=82.711,53.849,10.898,177.9740,12.3647,-1946.9339
C01041=83.875,52.589,10.937,178.1865,9.1389,-1947.9126
C01042=85.034,51.296,10.965,178.9987,6.1941,-1948.8999
C01043=86.364,49.571,10.978,179.6333,3.7272,-1950.1451
C01044=87.904,47.248,10.985,179.8919,1.7236,-1951.7422
C01045=89.436,44.606,10.991,179.9868,0.4356,-1953.4924
C01046=90.753,41.977,10.996,179.9977,0.0768,-1955.1775
C01047=91.870,39.492,11.000,179.9970,0.0075,-1956.7387
C01048=92.887,37.037,11.000,179.9968,0.0074,-1958.2613
C01049=93.854,34.490,10.996,179.9988,0.0798,-1959.8223
C01050=94.782,31.699,10.991,-179.9869,0.4366,-1961.5079
C01051=95.567,28.748,10.985,-179.8949,1.7218,-1963.2579
C01052=96.121,26.016,10.978,-179.6325,3.7259,-1964.8552
C01053=96.400,23.856,10.965,-178.9958,6.1937,-1966.1003
C01054=96.495,22.123,10.937,-178.1855,9.1378,-1967.0872
C01055=96.562,20.409,10.898,-177.9749,12.3697,-1968.0658
C01056=96.727,18.298,10.856,-178.5506,15.2200,-1969.2879
C01057=97.084,15.229,10.823,-179.4369,17.0680,-1971.0850
C01058=97.620,10.712,10.809,-179.9140,17.7316,-1973.7379
C01059=98.041,5.628,10.809,179.9935,17.7704,-1976.7146
C01060=98.204,0.000,10.809,180.0000,17.7591,-1980.0000
C01061=98.041,-5.628,10.809,-179.9935,17.7704,-1983.2854
C01062=97.620,-10.712,10.809,179.9140,17.7316,-1986.2621
C01063=97.084,-15.229,10.823,179.4369,17.0680,-1988.9150
C01064=96.727,-18.298,10.856,178.5506,15.2200,-1990.7121
C01065=96.562,-20.409,10.898,177.9749,12.3697,-1991.9342
C01066=96.495,-22.123,10.937,178.1855,9.1378,-1992.9128
C01067=96.400,-23.856,10.965,178.9958,6.1937,-1993.8997
C01068=96.121,-26.016,10.978,179.6325,3.7259,-1995.1448
C01069=95.567,-28.748,10.985,179.8949,1.7218,-1996.7421
C01070=94.782,-31.699,10.991,179.9869,0.4366,-1998.4921
C01071=93.854,-34.490,10.996,-179.9988,0.0798,-2000.1777
C01072=92.887,-37.037,11.000,-179.9968,0.0074,-2001.7387
C01073=91.870,-39.492,11.000,-179.9970,0.0075,-2003.2613
C01074=90.753,-41.977,10.996,-179.9977,0.0768,-2004.8225
C01075=89.436,-44.606,10.991,-179.9868,0.4356,-2006.5076
C01076=87.904,-47.248,10.985,-179.8919,1.7236,-2008.2578
C01077=86.364,-49.571,10.978,-179.6333,3.7272,-2009.8549
C01078=85.034,-51.296,10.965,-178.9987,6.1941,-2011.1001
C01079=83.875,-52.589,10.937,-178.1865,9.1389,-2012.0874
C01080=82.711,-53.849,10.898,-177.9740,12.3647,-2013.0661
C01081=81.334,-55.458,10.856,-178.5518,15.2206,-2014.2883
C01082=79.417,-57.880,10.823,-179.4413,17.0686,-2016.0850
C01083=76.603,-61.453,10.809,-179.9149,17.7331,-2018.7375
C01084=73.305,-65.346,10.809,179.9930,17.7700,-2021.7146
C01085=69.440,-69.440,10.809,-180.0000,17.7616,-2025.0000
C01086=65.346,-73.305,10.809,-179.9930,17.7700,-2028.2854
C01087=61.453,-76.603,10.809,179.9149,17.7331,-2031.2625
C01088=57.880,-79.417,10.823,179.4413,17.0686,-2033.9150
C01089=55.458,-81.334,10.856,178.5518,15.2206,-2035.7117
C01090=53.849,-82.711,10.898,177.9740,12.3647,-2036.9339
C01091=52.589,-83.875,10.937,178.1865,9.1389,-2037.9126
C01092=51.296,-85.034,10.965,178.9987,6.1941,-2038.8999
C01093=49.571,-86.364,10.978,179.6333,3.7272,-2040.1451
C01094=47.248,-87.904,10.985,179.8919,1.7236,-2041.7422
C01095=44.606,-89.436,10.991,179.9868,0.4356,-2043.4924
C01096=41.977,-90.753,10.996,179.9977,0.0768,-2045.1775
C01097=39.492,-91.870,11.000,179.9970,0.0075,-2046.7387
C01098=37.037,-92.887,11.000,179.9968,0.0074,-2048.2613
C01099=34.490,-93.854,10.996,179.9988,0.0798,-2049.8223
C01100=31.699,-94.782,10.991,-179.9869,0.4366,-2051.5079
C01101=28.748,-95.567,10.985,-179.8949,1.7218,-2053.2579
C01102=26.016,-96.121,10.978,-179.6325,3.7259,-2054.8552
C01103=23.856,-96.400,10.965,-178.9958,6.1937,-2056.1003
C01104=22.123,-96.495,10.937,-178.1855,9.1378,-2057.0872
C01105=20.409,-96.562,10.898,-177.9749,12.3697,-2058.0658
C01106=18.298,-96.727,10.856,-178.5506,15.2200,-2059.2879
C01107=15.229,-97.084,10.823,-179.4369,17.0680,-2061.0850
C01108=10.712,-97.620,10.809,-179.9140,17.7316,-2063.7379
C01109=5.628,-98.041,10.809,179.9935,17.7704,-2066.7146
C01110=0.000,-98.204,10.809,-180.0000,17.7591,-2070.0000
C01111=0.000,-98.204,10.809,-180.0000,17.7591,-2070.0000
C01112=-5.628,-98.041,10.809,-179.9935,17.7704,-2073.2854
C01113=-10.712,-97.620,10.809,179.9140,17.7316,-2076.2621
C01114=-15.229,-97.084,10.823,179.4369,17.0680,-2078.9150
C01115=-18.298,-96.727,10.856,178.5506,15.2200,-2080.7121
C01116=-20.409,-96.562,10.898,177.9749,12.3697,-2081.9342
C01117=-22.123,-96.495,10.937,178.1855,9.1378,-2082.9128
C01118=-23.856,-96.400,10.965,178.9958,6.1937,-2083.8997
C01119=-26.016,-96.121,10.978,179.6325,3.7259,-2085.1448
C01120=-28.748,-95.567,10.985,179.8949,1.7218,-2086.7421
C01121=-31.699,-94.782,10.991,179.9869,0.4366,-2088.4921
C01122=-34.490,-93.854,10.996,-179.9988,0.0798,-2090.1777
C01123=-37.037,-92.887,11.000,-179.9968,0.0074,-2091.7387
C01124=-39.492,-91.870,11.000,-179.9970,0.0075,-2093.2613
C01125=-41.977,-90.753,10.996,-179.9977,0.0768,-2094.8225
C01126=-44.606,-89.436,10.991,-179.9868,0.4356,-2096.5076
C01127=-47.248,-87.904,10.985,-179.8919,1.7236,-2098.2578
C01128=-49.571,-86.364,10.978,-179.6333,3.7272,-2099.8549
C01129=-51.296,-85.034,10.965,-178.9987,6.1941,-2101.1001
C01130=-52.589,-83.875,10.937,-178.1865,9.1389,-2102.0874
C01131=-53.849,-82.711,10.898,-177.9740,12.3647,-2103.0661
C01132=-55.458,-81.334,10.856,-178.5518,15.2206,-2104.2883
C01133=-57.880,-79.417,10.823,-179.4413,17.0686,-2106.0850
C01134=-61.453,-76.603,10.809,-179.9149,17.7331,-2108.7375
C01135=-65.346,-73.305,10.809,179.9930,17.7700,-2111.7146
C01136=-69.440,-69.440,10.809,180.0000,17.7616,-2115.0000
C01137=-73.305,-65.346,10.809,-179.9930,17.7700,-2118.2854
C01138=-76.603,-61.453,10.809,179.9149,17.7331,-2121.2625
C01139=-79.417,-57.880,10.823,179.4413,17.0686,-2123.9150
C01140=-81.334,-55.458,10.856,178.5518,15.2206,-2125.7117
C01141=-82.711,-53.849,10.898,177.9740,12.3647,-2126.9339
C01142=-83.875,-52.589,10.937,178.1865,9.1389,-2127.9126
C01143=-85.034,-51.296,10.965,178.9987,6.1941,-2128.8999
C01144=-86.364,-49.571,10.978,179.6333,3.7272,-2130.1451
C01145=-87.904,-47.248,10.985,179.8919,1.7236,-2131.7422
C01146=-89.436,-44.606,10.991,179.9868,0.4356,-2133.4924
C01147=-90.753,-41.977,10.996,179.9977,0.0768,-2135.1775
C01148=-91.870,-39.492,11.000,179.9970,0.0075,-2136.7387
C01149=-92.887,-37.037,11.000,179.9968,0.0074,-2138.2613
C01150=-93.854,-34.490,10.996,179.9988,0.0798,-2139.8223
C01151=-94.782,-31.699,10.991,-179.9869,0.4366,-2141.5079
C01152=-95.567,-28.748,10.985,-179.8949,1.7218,-2143.2579
C01153=-96.121,-26.016,10.978,-179.6325,3.7259,-2144.8552
C01154=-96.400,-23.856,10.965,-178.9958,6.1937,-2146.1003
C01155=-96.495,-22.123,10.937,-178.1855,9.1378,-2147.0872
C01156=-96.562,-20.409,10.898,-177.9749,12.3697,-2148.0658
C01157=-96.727,-18.298,10.856,-178.5506,15.2200,-2149.2879
C01158=-97.084,-15.229,10.823,-179.4369,17.0680,-2151.0850
C01159=-97.620,-10.712,10.809,-179.9140,17.7316,-2153.7379
C01160=-98.041,-5.628,10.809,179.9935,17.7704,-2156.7146
C01161=-98.204,0.000,10.809,-180.0000,17.7591,-2160.0000
C01162=-98.041,5.628,10.809,-179.9935,17.7704,-2163.2854
C01163=-97.620,10.712,10.809,179.9140,17.7316,-2166.2621
C01164=-97.084,15.229,10.823,179.4369,17.0680,-2168.9150
C01165=-96.727,18.298,10.856,178.5506,15.2200,-2170.7121
C01166=-96.562,20.409,10.898,177.9749,12.3697,-2171.9342
C01167=-96.495,22.123,10.937,178.1855,9.1378,-2172.9128
C01168=-96.400,23.856,10.965,178.9958,6.1937,-2173.8997
C01169=-96.121,26.016,10.978,179.6325,3.7259,-2175.1448
C01170=-95.567,28.748,10.985,179.8949,1.7218,-2176.7421
C01171=-94.782,31.699,10.991,179.9869,0.4366,-2178.4921
C01172=-93.854,34.490,10.996,-179.9988,0.0798,-2180.1777
C01173=-92.887,37.037,11.000,-179.9968,0.0074,-2181.7387
C01174=-91.870,39.492,11.000,-179.9970,0.0075,-2183.2613
C01175=-90.753,41.977,10.996,-179.9977,0.0768,-2184.8225
C01176=-89.436,44.606,10.991,-179.9868,0.4356,-2186.5076
C01177=-87.904,47.248,10.985,-179.8919,1.7236,-2188.2578
C01178=-86.364,49.571,10.978,-179.6333,3.7272,-2189.8549
C01179=-85.034,51.296,10.965,-178.9987,6.1941,-2191.1001
C01180=-83.875,52.589,10.937,-178.1865,9.1389,-2192.0874
C01181=-82.711,53.849,10.898,-177.9740,12.3647,-2193.0661
C01182=-81.334,55.458,10.856,-178.5518,15.2206,-2194.2883
C01183=-79.417,57.880,10.823,-179.4413,17.0686,-2196.0850
C01184=-76.603,61.453,10.809,-179.9149,17.7331,-2198.7375
C01185=-73.305,65.346,10.809,179.9930,17.7700,-2201.7146
C01186=-69.440,69.440,10.809,-180.0000,17.7616,-2205.0000
C01187=-65.346,73.305,10.809,-179.9930,17.7700,-2208.2854
C01188=-61.453,76.603,10.809,179.9149,17.7331,-2211.2625
C01189=-57.880,79.417,10.823,179.4413,17.0686,-2213.9150
C01190=-55.458,81.334,10.856,178.5518,15.2206,-2215.7117
C01191=-53.849,82.711,10.898,177.9740,12.3647,-2216.9339
C01192=-52.589,83.875,10.937,178.1865,9.1389,-2217.9126
C01193=-51.296,85.034,10.965,178.9987,6.1941,-2218.8999
C01194=-49.571,86.364,10.978,179.6333,3.7272,-2220.1451
C01195=-47.248,87.904,10.985,179.8919,1.7236,-2221.7422
C01196=-44.606,89.436,10.991,179.9868,0.4356,-2223.4924
C01197=-41.977,90.753,10.996,179.9977,0.0768,-2225.1775
C01198=-39.492,91.870,11.000,179.9970,0.0075,-2226.7387
C01199=-37.037,92.887,11.000,179.9968,0.0074,-2228.2613
C01200=-34.490,93.854,10.996,179.9988,0.0798,-2229.8223
C01201=-31.699,94.782,10.991,-179.9869,0.4366,-2231.5079
C01202=-28.748,95.567,10.985,-179.8949,1.7218,-2233.2579
C01203=-26.016,96.121,10.978,-179.6325,3.7259,-2234.8552
C01204=-23.856,96.400,10.965,-178.9958,6.1937,-2236.1003
C01205=-22.123,96.495,10.937,-178.1855,9.1378,-2237.0872
C01206=-20.409,96.562,10.898,-177.9749,12.3697,-2238.0658
C01207=-18.298,96.727,10.856,-178.5506,15.2200,-2239.2879
C01208=-15.229,97.084,10.823,-179.4369,17.0680,-2241.0850
C01209=-10.712,97.620,10.809,-179.9140,17.7316,-2243.7379
C01210=-5.628,98.041,10.809,179.9935,17.7704,-2246.7146
C01211=0.000,98.204,10.809,180.0000,17.7591,-2250.0000
C01212=0.000,97.482,12.888,180.0000,20.4756,-2250.0000
C01213=5.562,97.322,12.887,-179.9859,20.4854,-2253.2709
C01214=10.602,96.908,12.888,179.8598,20.4405,-2256.2435
C01215=15.094,96.401,12.910,179.0729,19.6670,-2258.8988
C01216=18.135,96.115,12.963,177.6149,17.4078,-2260.6850
C01217=20.227,96.057,13.031,176.7212,13.8489,-2261.8912
C01218=21.929,96.117,13.096,177.1319,9.9912,-2262.8520
C01219=23.652,96.157,13.142,178.4135,6.7582,-2263.8189
C01220=25.795,96.000,13.164,179.4239,4.0853,-2265.0400
C01221=28.540,95.542,13.175,179.8391,1.8598,-2266.6318
C01222=31.535,94.812,13.184,179.9785,0.4457,-2268.3974
C01223=34.387,93.888,13.193,-179.9987,0.0798,-2270.1155
C01224=37.002,92.901,13.199,-179.9989,0.0128,-2271.7171
C01225=39.526,91.855,13.199,-179.9993,0.0128,-2273.2826
C01226=42.074,90.704,13.193,179.9998,0.0820,-2274.8847
C01227=44.743,89.341,13.184,-179.9798,0.4459,-2276.6022
C01228=47.377,87.740,13.175,-179.8379,1.8589,-2278.3677
C01229=49.643,86.123,13.164,-179.4219,4.0858,-2279.9600
C01230=51.269,84.717,13.142,-178.4147,6.7570,-2281.1815
C01231=52.459,83.471,13.096,-177.1286,9.9939,-2282.1481
C01232=53.620,82.225,13.031,-176.7209,13.8526,-2283.1089
C01233=55.140,80.787,12.963,-177.6104,17.4102,-2284.3149
C01234=57.492,78.839,12.910,-179.0715,19.6676,-2286.1008
C01235=61.028,76.021,12.888,-179.8604,20.4407,-2288.7567
C01236=64.884,72.750,12.887,179.9887,20.4843,-2291.7290
C01237=68.930,68.930,12.888,-180.0000,20.4721,-2295.0000
C01238=72.750,64.884,12.887,-179.9887,20.4843,-2298.2710
C01239=76.021,61.028,12.888,179.8604,20.4407,-2301.2433
C01240=78.839,57.492,12.910,179.0715,19.6676,-2303.8992
C01241=80.787,55.140,12.963,177.6104,17.4102,-2305.6851
C01242=82.225,53.620,13.031,176.7209,13.8526,-2306.8911
C01243=83.471,52.459,13.096,177.1286,9.9939,-2307.8519
C01244=84.717,51.269,13.142,178.4147,6.7570,-2308.8185
C01245=86.123,49.643,13.164,179.4219,4.0858,-2310.0400
C01246=87.740,47.377,13.175,179.8379,1.8589,-2311.6323
C01247=89.341,44.743,13.184,179.9798,0.4459,-2313.3978
C01248=90.704,42.074,13.193,-179.9998,0.0820,-2315.1153
C01249=91.855,39.526,13.199,179.9993,0.0128,-2316.7174
C01250=92.901,37.002,13.199,179.9989,0.0128,-2318.2829
C01251=93.888,34.387,13.193,179.9987,0.0798,-2319.8845
C01252=94.812,31.535,13.184,-179.9785,0.4457,-2321.6026
C01253=95.542,28.540,13.175,-179.8391,1.8598,-2323.3682
C01254=96.000,25.795,13.164,-179.4239,4.0853,-2324.9600
C01255=96.157,23.652,13.142,-178.4135,6.7582,-2326.1811
C01256=96.117,21.929,13.096,-177.1319,9.9912,-2327.1480
C01257=96.057,20.227,13.031,-176.7212,13.8489,-2328.1088
C01258=96.115,18.135,12.963,-177.6149,17.4078,-2329.3150
C01259=96.401,15.094,12.910,-179.0729,19.6670,-2331.1012
C01260=96.908,10.602,12.888,-179.8598,20.4405,-2333.7565
C01261=97.322,5.562,12.887,179.9859,20.4854,-2336.7291
C01262=97.482,0.000,12.888,180.0000,20.4756,-2340.0000
C01263=97.322,-5.562,12.887,-179.9859,20.4854,-2343.2709
C01264=96.908,-10.602,12.888,179.8598,20.4405,-2346.2435
C01265=96.401,-15.094,12.910,179.0729,19.6670,-2348.8988
C01266=96.115,-18.135,12.963,177.6149,17.4078,-2350.6850
C01267=96.057,-20.227,13.031,176.7212,13.8489,-2351.8912
C01268=96.117,-21.929,13.096,177.1319,9.9912,-2352.8520
C01269=96.157,-23.652,13.142,178.4135,6.7582,-2353.8189
C01270=96.000,-25.795,13.164,179.4239,4.0853,-2355.0400
C01271=95.542,-28.540,13.175,179.8391,1.8598,-2356.6318
C01272=94.812,-31.535,13.184,179.9785,0.4457,-2358.3974
C01273=93.888,-34.387,13.193,-179.9987,0.0798,-2360.1155
C01274=92.901,-37.002,13.199,-179.9989,0.0128,-2361.7171
C01275=91.855,-39.526,13.199,-179.9993,0.0128,-2363.2826
C01276=90.704,-42.074,13.193,179.9998,0.0820,-2364.8847
C01277=89.341,-44.743,13.184,-179.9798,0.4459,-2366.6022
C01278=87.740,-47.377,13.175,-179.8379,1.8589,-2368.3677
C01279=86.123,-49.643,13.164,-179.4219,4.0858,-2369.9600
C01280=84.717,-51.269,13.142,-178.4147,6.7570,-2371.1815
C01281=83.471,-52.459,13.096,-177.1286,9.9939,-2372.1481
C01282=82.225,-53.620,13.031,-176.7209,13.8526,-2373.1089
C01283=80.787,-55.140,12.963,-177.6104,17.4102,-2374.3149
C01284=78.839,-57.492,12.910,-179.0715,19.6676,-2376.1008
C01285=76.021,-61.028,12.888,-179.8604,20.4407,-2378.7567
C01286=72.750,-64.884,12.887,179.9887,20.4843,-2381.7290
C01287=68.930,-68.930,12.888,-180.0000,20.4721,-2385.0000
C01288=64.884,-72.750,12.887,-179.9887,20.4843,-2388.2710
C01289=61.028,-76.021,12.888,179.8604,20.4407,-2391.2433
C01290=57.492,-78.839,12.910,179.0715,19.6676,-2393.8992
C01291=55.140,-80.787,12.963,177.6104,17.4102,-2395.6851
C01292=53.620,-82.225,13.031,176.7209,13.8526,-2396.8911
C01293=52.459,-83.471,13.096,177.1286,9.9939,-2397.8519
C01294=51.269,-84.717,13.142,178.4147,6.7570,-2398.8185
C01295=49.643,-86.123,13.164,179.4219,4.0858,-2400.0400
C01296=47.377,-87.740,13.175,179.8379,1.8589,-2401.6323
C01297=44.743,-89.341,13.184,179.9798,0.4459,-2403.3978
C01298=42.074,-90.704,13.193,-179.9998,0.0820,-2405.1153
C01299=39.526,-91.855,13.199,179.9993,0.0128,-2406.7174
C01300=37.002,-92.901,13.199,179.9989,0.0128,-2408.2829
C01301=34.387,-93.888,13.193,179.9987,0.0798,-2409.8845
C01302=31.535,-94.812,13.184,-179.9785,0.4457,-2411.6026
C01303=28.540,-95.542,13.175,-179.8391,1.8598,-2413.3682
C01304=25.795,-96.000,13.164,-179.4239,4.0853,-2414.9600
C01305=23.652,-96.157,13.142,-178.4135,6.7582,-2416.1811
C01306=21.929,-96.117,13.096,-177.1319,9.9912,-2417.1480
C01307=20.227,-96.057,13.031,-176.7212,13.8489,-2418.1088
C01308=18.135,-96.115,12.963,-177.6149,17.4078,-2419.3150
C01309=15.094,-96.401,12.910,-179.0729,19.6670,-2421.1012
C01310=10.602,-96.908,12.888,-179.8598,20.4405,-2423.7565
C01311=5.562,-97.322,12.887,179.9859,20.4854,-2426.7291
C01312=0.000,-97.482,12.888,-180.0000,20.4756,-2430.0000
C01313=0.000,-97.482,12.888,-180.0000,20.4756,-2430.0000
C01314=-5.562,-97.322,12.887,-179.9859,20.4854,-2433.2709
C01315=-10.602,-96.908,12.888,179.8598,20.4405,-2436.2435
C01316=-15.094,-96.401,12.910,179.0729,19.6670,-2438.8988
C01317=-18.135,-96.115,12.963,177.6149,17.4078,-2440.6850
C01318=-20.227,-96.057,13.031,176.7212,13.8489,-2441.8912
C01319=-21.929,-96.117,13.096,177.1319,9.9912,-2442.8520
C01320=-23.652,-96.157,13.142,178.4135,6.7582,-2443.8189
C01321=-25.795,-96.000,13.164,179.4239,4.0853,-2445.0400
C01322=-28.540,-95.542,13.175,179.8391,1.8598,-2446.6318
C01323=-31.535,-94.812,13.184,179.9785,0.4457,-2448.3974
C01324=-34.387,-93.888,13.193,-179.9987,0.0798,-2450.1155
C01325=-37.002,-92.901,13.199,-179.9989,0.0128,-2451.7171
C01326=-39.526,-91.855,13.199,-179.9993,0.0128,-2453.2826
C01327=-42.074,-90.704,13.193,179.9998,0.0820,-2454.8847
C01328=-44.743,-89.341,13.184,-179.9798,0.4459,-2456.6022
C01329=-47.377,-87.740,13.175,-179.8379,1.8589,-2458.3677
C01330=-49.643,-86.123,13.164,-179.4219,4.0858,-2459.9600
C01331=-51.269,-84.717,13.142,-178.4147,6.7570,-2461.1815
C01332=-52.459,-83.471,13.096,-177.1286,9.9939,-2462.1481
C01333=-53.620,-82.225,13.031,-176.7209,13.8526,-2463.1089
C01334=-55.140,-80.787,12.963,-177.6104,17.4102,-2464.3149
C01335=-57.492,-78.839,12.910,-179.0715,19.6676,-2466.1008
C01336=-61.028,-76.021,12.888,-179.8604,20.4407,-2468.7567
C01337=-64.884,-72.750,12.887,179.9887,20.4843,-2471.7290
C01338=-68.930,-68.930,12.888,180.0000,20.4721,-2475.0000
C01339=-72.750,-64.884,12.887,-179.9887,20.4843,-2478.2710
C01340=-76.021,-61.028,12.888,179.8604,20.4407,-2481.2433
C01341=-78.839,-57.492,12.910,179.0715,19.6676,-2483.8992
C01342=-80.787,-55.140,12.963,177.6104,17.4102,-2485.6851
C01343=-82.225,-53.620,13.031,176.7209,13.8526,-2486.8911
C01344=-83.471,-52.459,13.096,177.1286,9.9939,-2487.8519
C01345=-84.717,-51.269,13.142,178.4147,6.7570,-2488.8185
C01346=-86.123,-49.643,13.164,179.4219,4.0858,-2490.0400
C01347=-87.740,-47.377,13.175,179.8379,1.8589,-2491.6323
C01348=-89.341,-44.743,13.184,179.9798,0.4459,-2493.3978
C01349=-90.704,-42.074,13.193,-179.9998,0.0820,-2495.1153
C01350=-91.855,-39.526,13.199,179.9993,0.0128,-2496.7174
C01351=-92.901,-37.002,13.199,179.9989,0.0128,-2498.2829
C01352=-93.888,-34.387,13.193,179.9987,0.0798,-2499.8845
C01353=-94.812,-31.535,13.184,-179.9785,0.4457,-2501.6026
C01354=-95.542,-28.540,13.175,-179.8391,1.8598,-2503.3682
C01355=-96.000,-25.795,13.164,-179.4239,4.0853,-2504.9600
C01356=-96.157,-23.652,13.142,-178.4135,6.7582,-2506.1811
C01357=-96.117,-21.929,13.096,-177.1319,9.9912,-2507.1480
C01358=-96.057,-20.227,13.031,-176.7212,13.8489,-2508.1088
C01359=-96.115,-18.135,12.963,-177.6149,17.4078,-2509.3150
C01360=-96.401,-15.094,12.910,-179.0729,19.6670,-2511.1012
C01361=-96.908,-10.602,12.888,-179.8598,20.4405,-2513.7565
C01362=-97.322,-5.562,12.887,179.9859,20.4854,-2516.7291
C01363=-97.482,0.000,12.888,-180.0000,20.4756,-2520.0000
C01364=-97.322,5.562,12.887,-179.9859,20.4854,-2523.2709
C01365=-96.908,10.602,12.888,179.8598,20.4405,-2526.2435
C01366=-96.401,15.094,12.910,179.0729,19.6670,-2528.8988
C01367=-96.115,18.135,12.963,177.6149,17.4078,-2530.6850
C01368=-96.057,20.227,13.031,176.7212,13.8489,-2531.8912
C01369=-96.117,21.929,13.096,177.1319,9.9912,-2532.8520
C01370=-96.157,23.652,13.142,178.4135,6.7582,-2533.8189
C01371=-96.000,25.795,13.164,179.4239,4.0853,-2535.0400
C01372=-95.542,28.540,13.175,179.8391,1.8598,-2536.6318
C01373=-94.812,31.535,13.184,179.9785,0.4457,-2538.3974
C01374=-93.888,34.387,13.193,-179.9987,0.0798,-2540.1155
C01375=-92.901,37.002,13.199,-179.9989,0.0128,-2541.7171
C01376=-91.855,39.526,13.199,-179.9993,0.0128,-2543.2826
C01377=-90.704,42.074,13.193,179.9998,0.0820,-2544.8847
C01378=-89.341,44.743,13.184,-179.9798,0.4459,-2546.6022
C01379=-87.740,47.377,13.175,-179.8379,1.8589,-2548.3677
C01380=-86.123,49.643,13.164,-179.4219,4.0858,-2549.9600
C01381=-84.717,51.269,13.142,-178.4147,6.7570,-2551.1815
C01382=-83.471,52.459,13.096,-177.1286,9.9939,-2552.1481
C01383=-82.225,53.620,13.031,-176.7209,13.8526,-2553.1089
C01384=-80.787,55.140,12.963,-177.6104,17.4102,-2554.3149
C01385=-78.839,57.492,12.910,-179.0715,19.6676,-2556.1008
C01386=-76.021,61.028,12.888,-179.8604,20.4407,-2558.7567
C01387=-72.750,64.884,12.887,179.9887,20.4843,-2561.7290
C01388=-68.930,68.930,12.888,180.0000,20.4721,-2565.0000
C01389=-64.884,72.750,12.887,-179.9887,20.4843,-2568.2710
C01390=-61.028,76.021,12.888,179.8604,20.4407,-2571.2433
C01391=-57.492,78.839,12.910,179.0715,19.6676,-2573.8992
C01392=-55.140,80.787,12.963,177.6104,17.4102,-2575.6851
C01393=-53.620,82.225,13.031,176.7209,13.8526,-2576.8911
C01394=-52.459,83.471,13.096,177.1286,9.9939,-2577.8519
C01395=-51.269,84.717,13.142,178.4147,6.7570,-2578.8185
C01396=-49.643,86.123,13.164,179.4219,4.0858,-2580.0400
C01397=-47.377,87.740,13.175,179.8379,1.8589,-2581.6323
C01398=-44.743,89.341,13.184,179.9798,0.4459,-2583.3978
C01399=-42.074,90.704,13.193,-179.9998,0.0820,-2585.1153
C01400=-39.526,91.855,13.199,179.9993,0.0128,-2586.7174
C01401=-37.002,92.901,13.199,179.9989,0.0128,-2588.2829
C01402=-34.387,93.888,13.193,179.9987,0.0798,-2589.8845
C01403=-31.535,94.812,13.184,-179.9785,0.4457,-2591.6026
C01404=-28.540,95.542,13.175,-179.8391,1.8598,-2593.3682
C01405=-25.795,96.000,13.164,-179.4239,4.0853,-2594.9600
C01406=-23.652,96.157,13.142,-178.4135,6.7582,-2596.1811
C01407=-21.929,96.117,13.096,-177.1319,9.9912,-2597.1480
C01408=-20.227,96.057,13.031,-176.7212,13.8489,-2598.1088
C01409=-18.135,96.115,12.963,-177.6149,17.4078,-2599.3150
C01410=-15.094,96.401,12.910,-179.0729,19.6670,-2601.1012
C01411=-10.602,96.908,12.888,-179.8598,20.4405,-2603.7565
C01412=-5.562,97.322,12.887,179.9859,20.4854,-2606.7291
C01413=0.000,97.482,12.888,180.0000,20.4756,-2610.0000
C01414=0.000,96.668,14.931,180.0000,22.9187,-2610.0000
C01415=5.488,96.511,14.930,-179.9826,22.9316,-2613.2546
C01416=10.476,96.104,14.932,179.7920,22.8765,-2616.2211
C01417=14.942,95.628,14.964,178.5991,21.9924,-2618.8807
C01418=17.951,95.422,15.043,176.3980,19.2373,-2620.6541
C01419=20.020,95.481,15.144,175.2071,14.8082,-2621.8420
C01420=21.708,95.685,15.242,175.9369,10.3073,-2622.7823
C01421=23.417,95.878,15.312,177.7556,6.9686,-2623.7251
C01422=25.541,95.862,15.345,179.1830,4.2642,-2624.9190
C01423=28.302,95.513,15.362,179.7758,1.9061,-2626.5054
C01424=31.347,94.846,15.376,179.9757,0.4204,-2628.2889
C01425=34.268,93.927,15.390,179.9994,0.0852,-2630.0438
C01426=36.962,92.916,15.399,-179.9989,0.0128,-2631.6927
C01427=39.566,91.838,15.399,-179.9993,0.0128,-2633.3075
C01428=42.186,90.648,15.390,179.9997,0.0820,-2634.9564
C01429=44.901,89.232,15.376,-179.9729,0.4177,-2636.7113
C01430=47.525,87.551,15.362,-179.7770,1.9077,-2638.4943
C01431=49.724,85.845,15.345,-179.1812,4.2648,-2640.0807
C01432=51.237,84.354,15.312,-177.7577,6.9647,-2641.2747
C01433=52.309,83.010,15.242,-175.9409,10.3085,-2642.2172
C01434=53.359,81.672,15.144,-175.2066,14.8105,-2643.1579
C01435=54.780,80.167,15.043,-176.4009,19.2366,-2644.3457
C01436=57.054,78.185,14.964,-178.6006,21.9938,-2646.1194
C01437=60.548,75.364,14.932,-179.7889,22.8755,-2648.7787
C01438=64.363,72.124,14.930,179.9816,22.9306,-2651.7455
C01439=68.355,68.355,14.931,-180.0000,22.9226,-2655.0000
C01440=72.124,64.363,14.930,-179.9816,22.9306,-2658.2545
C01441=75.364,60.548,14.932,179.7889,22.8755,-2661.2213
C01442=78.185,57.054,14.964,178.6006,21.9938,-2663.8806
C01443=80.167,54.780,15.043,176.4009,19.2366,-2665.6543
C01444=81.672,53.359,15.144,175.2066,14.8105,-2666.8421
C01445=83.010,52.309,15.242,175.9409,10.3085,-2667.7828
C01446=84.354,51.237,15.312,177.7577,6.9647,-2668.7253
C01447=85.845,49.724,15.345,179.1812,4.2648,-2669.9193
C01448=87.551,47.525,15.362,179.7770,1.9077,-2671.5057
C01449=89.232,44.901,15.376,179.9729,0.4177,-2673.2887
C01450=90.648,42.186,15.390,-179.9997,0.0820,-2675.0436
C01451=91.838,39.566,15.399,179.9993,0.0128,-2676.6925
C01452=92.916,36.962,15.399,179.9989,0.0128,-2678.3073
C01453=93.927,34.268,15.390,-179.9994,0.0852,-2679.9562
C01454=94.846,31.347,15.376,-179.9757,0.4204,-2681.7111
C01455=95.513,28.302,15.362,-179.7758,1.9061,-2683.4946
C01456=95.862,25.541,15.345,-179.1830,4.2642,-2685.0810
C01457=95.878,23.417,15.312,-177.7556,6.9686,-2686.2749
C01458=95.685,21.708,15.242,-175.9369,10.3073,-2687.2177
C01459=95.481,20.020,15.144,-175.2071,14.8082,-2688.1580
C01460=95.422,17.951,15.043,-176.3980,19.2373,-2689.3459
C01461=95.628,14.942,14.964,-178.5991,21.9924,-2691.1193
C01462=96.104,10.476,14.932,-179.7920,22.8765,-2693.7789
C01463=96.511,5.488,14.930,179.9826,22.9316,-2696.7454
C01464=96.668,0.000,14.931,180.0000,22.9187,-2700.0000
C01465=96.511,-5.488,14.930,-179.9826,22.9316,-2703.2546
C01466=96.104,-10.476,14.932,179.7920,22.8765,-2706.2211
C01467=95.628,-14.942,14.964,178.5991,21.9924,-2708.8807
C01468=95.422,-17.951,15.043,176.3980,19.2373,-2710.6541
C01469=95.481,-20.020,15.144,175.2071,14.8082,-2711.8420
C01470=95.685,-21.708,15.242,175.9369,10.3073,-2712.7823
C01471=95.878,-23.417,15.312,177.7556,6.9686,-2713.7251
C01472=95.862,-25.541,15.345,179.1830,4.2642,-2714.9190
C01473=95.513,-28.302,15.362,179.7758,1.9061,-2716.5054
C01474=94.846,-31.347,15.376,179.9757,0.4204,-2718.2889
C01475=93.927,-34.268,15.390,179.9994,0.0852,-2720.0438
C01476=92.916,-36.962,15.399,-179.9989,0.0128,-2721.6927
C01477=91.838,-39.566,15.399,-179.9993,0.0128,-2723.3075
C01478=90.648,-42.186,15.390,179.9997,0.0820,-2724.9564
C01479=89.232,-44.901,15.376,-179.9729,0.4177,-2726.7113
C01480=87.551,-47.525,15.362,-179.7770,1.9077,-2728.4943
C01481=85.845,-49.724,15.345,-179.1812,4.2648,-2730.0807
C01482=84.354,-51.237,15.312,-177.7577,6.9647,-2731.2747
C01483=83.010,-52.309,15.242,-175.9409,10.3085,-2732.2172
C01484=81.672,-53.359,15.144,-175.2066,14.8105,-2733.1579
C01485=80.167,-54.780,15.043,-176.4009,19.2366,-2734.3457
C01486=78.185,-57.054,14.964,-178.6006,21.9938,-2736.1194
C01487=75.364,-60.548,14.932,-179.7889,22.8755,-2738.7787
C01488=72.124,-64.363,14.930,179.9816,22.9306,-2741.7455
C01489=68.355,-68.355,14.931,-180.0000,22.9226,-2745.0000
C01490=64.363,-72.124,14.930,-179.9816,22.9306,-2748.2545
C01491=60.548,-75.364,14.932,179.7889,22.8755,-2751.2213
C01492=57.054,-78.185,14.964,178.6006,21.9938,-2753.8806
C01493=54.780,-80.167,15.043,176.4009,19.2366,-2755.6543
C01494=53.359,-81.672,15.144,175.2066,14.8105,-2756.8421
C01495=52.309,-83.010,15.242,175.9409,10.3085,-2757.7828
C01496=51.237,-84.354,15.312,177.7577,6.9647,-2758.7253
C01497=49.724,-85.845,15.345,179.1812,4.2648,-2759.9193
C01498=47.525,-87.551,15.362,179.7770,1.9077,-2761.5057
C01499=44.901,-89.232,15.376,179.9729,0.4177,-2763.2887
C01500=42.186,-90.648,15.390,-179.9997,0.0820,-2765.0436
C01501=39.566,-91.838,15.399,179.9993,0.0128,-2766.6925
C01502=36.962,-92.916,15.399,179.9989,0.0128,-2768.3073
C01503=34.268,-93.927,15.390,-179.9994,0.0852,-2769.9562
C01504=31.347,-94.846,15.376,-179.9757,0.4204,-2771.7111
C01505=28.302,-95.513,15.362,-179.7758,1.9061,-2773.4946
C01506=25.541,-95.862,15.345,-179.1830,4.2642,-2775.0810
C01507=23.417,-95.878,15.312,-177.7556,6.9686,-2776.2749
C01508=21.708,-95.685,15.242,-175.9369,10.3073,-2777.2177
C01509=20.020,-95.481,15.144,-175.2071,14.8082,-2778.1580
C01510=17.951,-95.422,15.043,-176.3980,19.2373,-2779.3459
C01511=14.942,-95.628,14.964,-178.5991,21.9924,-2781.1193
C01512=10.476,-96.104,14.932,-179.7920,22.8765,-2783.7789
C01513=5.488,-96.511,14.930,179.9826,22.9316,-2786.7454
C01514=0.000,-96.668,14.931,-180.0000,22.9187,-2790.0000
C01515=0.000,-96.668,14.931,-180.0000,22.9187,-2790.0000
C01516=-5.488,-96.511,14.930,-179.9826,22.9316,-2793.2546
C01517=-10.476,-96.104,14.932,179.7920,22.8765,-2796.2211
C01518=-14.942,-95.628,14.964,178.5991,21.9924,-2798.8807
C01519=-17.951,-95.422,15.043,176.3980,19.2373,-2800.6541
C01520=-20.020,-95.481,15.144,175.2071,14.8082,-2801.8420
C01521=-21.708,-95.685,15.242,175.9369,10.3073,-2802.7823
C01522=-23.417,-95.878,15.312,177.7556,6.9686,-2803.7251
C01523=-25.541,-95.862,15.345,179.1830,4.2642,-2804.9190
C01524=-28.302,-95.513,15.362,179.7758,1.9061,-2806.5054
C01525=-31.347,-94.846,15.376,179.9757,0.4204,-2808.2889
C01526=-34.268,-93.927,15.390,179.9994,0.0852,-2810.0438
C01527=-36.962,-92.916,15.399,-179.9989,0.0128,-2811.6927
C01528=-39.566,-91.838,15.399,-179.9993,0.0128,-2813.3075
C01529=-42.186,-90.648,15.390,179.9997,0.0820,-2814.9564
C01530=-44.901,-89.232,15.376,-179.9729,0.4177,-2816.7113
C01531=-47.525,-87.551,15.362,-179.7770,1.9077,-2818.4943
C01532=-49.724,-85.845,15.345,-179.1812,4.2648,-2820.0807
C01533=-51.237,-84.354,15.312,-177.7577,6.9647,-2821.2747
C01534=-52.309,-83.010,15.242,-175.9409,10.3085,-2822.2172
C01535=-53.359,-81.672,15.144,-175.2066,14.8105,-2823.1579
C01536=-54.780,-80.167,15.043,-176.4009,19.2366,-2824.3457
C01537=-57.054,-78.185,14.964,-178.6006,21.9938,-2826.1194
C01538=-60.548,-75.364,14.932,-179.7889,22.8755,-2828.7787
C01539=-64.363,-72.124,14.930,179.9816,22.9306,-2831.7455
C01540=-68.355,-68.355,14.931,180.0000,22.9226,-2835.0000
C01541=-72.124,-64.363,14.930,-179.9816,22.9306,-2838.2545
C01542=-75.364,-60.548,14.932,179.7889,22.8755,-2841.2213
C01543=-78.185,-57.054,14.964,178.6006,21.9938,-2843.8806
C01544=-80.167,-54.780,15.043,176.4009,19.2366,-2845.6543
C01545=-81.672,-53.359,15.144,175.2066,14.8105,-2846.8421
C01546=-83.010,-52.309,15.242,175.9409,10.3085,-2847.7828
C01547=-84.354,-51.237,15.312,177.7577,6.9647,-2848.7253
C01548=-85.845,-49.724,15.345,179.1812,4.2648,-2849.9193
C01549=-87.551,-47.525,15.362,179.7770,1.9077,-2851.5057
C01550=-89.232,-44.901,15.376,179.9729,0.4177,-2853.2887
C01551=-90.648,-42.186,15.390,-179.9997,0.0820,-2855.0436
C01552=-91.838,-39.566,15.399,179.9993,0.0128,-2856.6925
C01553=-92.916,-36.962,15.399,179.9989,0.0128,-2858.3073
C01554=-93.927,-34.268,15.390,-179.9994,0.0852,-2859.9562
C01555=-94.846,-31.347,15.376,-179.9757,0.4204,-2861.7111
C01556=-95.513,-28.302,15.362,-179.7758,1.9061,-2863.4946
C01557=-95.862,-25.541,15.345,-179.1830,4.2642,-2865.0810
C01558=-95.878,-23.417,15.312,-177.7556,6.9686,-2866.2749
C01559=-95.685,-21.708,15.242,-175.9369,10.3073,-2867.2177
C01560=-95.481,-20.020,15.144,-175.2071,14.8082,-2868.1580
C01561=-95.422,-17.951,15.043,-176.3980,19.2373,-2869.3459
C01562=-95.628,-14.942,14.964,-178.5991,21.9924,-2871.1193
C01563=-96.104,-10.476,14.932,-179.7920,22.8765,-2873.7789
C01564=-96.511,-5.488,14.930,179.9826,22.9316,-2876.7454
C01565=-96.668,0.000,14.931,-180.0000,22.9187,-2880.0000
C01566=-96.511,5.488,14.930,-179.9826,22.9316,-2883.2546
C01567=-96.104,10.476,14.932,179.7920,22.8765,-2886.2211
C01568=-95.628,14.942,14.964,178.5991,21.9924,-2888.8807
C01569=-95.422,17.951,15.043,176.3980,19.2373,-2890.6541
C01570=-95.481,20.020,15.144,175.2071,14.8082,-2891.8420
C01571=-95.685,21.708,15.242,175.9369,10.3073,-2892.7823
C01572=-95.878,23.417,15.312,177.7556,6.9686,-2893.7251
C01573=-95.862,25.541,15.345,179.1830,4.2642,-2894.9190
C01574=-95.513,28.302,15.362,179.7758,1.9061,-2896.5054
C01575=-94.846,31.347,15.376,179.9757,0.4204,-2898.2889
C01576=-93.927,34.268,15.390,179.9994,0.0852,-2900.0438
C01577=-92.916,36.962,15.399,-179.9989,0.0128,-2901.6927
C01578=-91.838,39.566,15.399,-179.9993,0.0128,-2903.3075
C01579=-90.648,42.186,15.390,179.9997,0.0820,-2904.9564
C01580=-89.232,44.901,15.376,-179.9729,0.4177,-2906.7113
C01581=-87.551,47.525,15.362,-179.7770,1.9077,-2908.4943
C01582=-85.845,49.724,15.345,-179.1812,4.2648,-2910.0807
C01583=-84.354,51.237,15.312,-177.7577,6.9647,-2911.2747
C01584=-83.010,52.309,15.242,-175.9409,10.3085,-2912.2172
C01585=-81.672,53.359,15.144,-175.2066,14.8105,-2913.1579
C01586=-80.167,54.780,15.043,-176.4009,19.2366,-2914.3457
C01587=-78.185,57.054,14.964,-178.6006,21.9938,-2916.1194
C01588=-75.364,60.548,14.932,-179.7889,22.8755,-2918.7787
C01589=-72.124,64.363,14.930,179.9816,22.9306,-2921.7455
C01590=-68.355,68.355,14.931,180.0000,22.9226,-2925.0000
C01591=-64.363,72.124,14.930,-179.9816,22.9306,-2928.2545
C01592=-60.548,75.364,14.932,179.7889,22.8755,-2931.2213
C01593=-57.054,78.185,14.964,178.6006,21.9938,-2933.8806
C01594=-54.780,80.167,15.043,176.4009,19.2366,-2935.6543
C01595=-53.359,81.672,15.144,175.2066,14.8105,-2936.8421
C01596=-52.309,83.010,15.242,175.9409,10.3085,-2937.7828
C01597=-51.237,84.354,15.312,177.7577,6.9647,-2938.7253
C01598=-49.724,85.845,15.345,179.1812,4.2648,-2939.9193
C01599=-47.525,87.551,15.362,179.7770,1.9077,-2941.5057
C01600=-44.901,89.232,15.376,179.9729,0.4177,-2943.2887
C01601=-42.186,90.648,15.390,-179.9997,0.0820,-2945.0436
C01602=-39.566,91.838,15.399,179.9993,0.0128,-2946.6925
C01603=-36.962,92.916,15.399,179.9989,0.0128,-2948.3073
C01604=-34.268,93.927,15.390,-179.9994,0.0852,-2949.9562
C01605=-31.347,94.846,15.376,-179.9757,0.4204,-2951.7111
C01606=-28.302,95.513,15.362,-179.7758,1.9061,-2953.4946
C01607=-25.541,95.862,15.345,-179.1830,4.2642,-2955.0810
C01608=-23.417,95.878,15.312,-177.7556,6.9686,-2956.2749
C01609=-21.708,95.685,15.242,-175.9369,10.3073,-2957.2177
C01610=-20.020,95.481,15.144,-175.2071,14.8082,-2958.1580
C01611=-17.951,95.422,15.043,-176.3980,19.2373,-2959.3459
C01612=-14.942,95.628,14.964,-178.5991,21.9924,-2961.1193
C01613=-10.476,96.104,14.932,-179.7920,22.8765,-2963.7789
C01614=-5.488,96.511,14.930,179.9826,22.9316,-2966.7454
C01615=0.000,96.668,14.931,-180.0000,22.9187,-2970.0000
C01616=0.000,95.772,16.941,-180.0000,25.1121,-2970.0000
C01617=5.406,95.617,16.939,-179.9726,25.1250,-2973.2359
C01618=10.339,95.219,16.941,179.6989,25.0665,-2976.1970
C01619=14.774,94.777,16.986,178.0084,24.0583,-2978.8601
C01620=17.748,94.656,17.095,174.9374,20.6589,-2980.6197
C01621=19.790,94.842,17.237,173.5645,15.1715,-2981.7864
C01622=21.462,95.203,17.374,174.7852,10.0480,-2982.7041
C01623=23.155,95.565,17.473,177.1151,6.7819,-2983.6200
C01624=25.257,95.708,17.521,178.9370,4.2461,-2984.7831
C01625=28.035,95.481,17.545,179.7194,1.8706,-2986.3632
C01626=31.135,94.884,17.565,179.9727,0.3589,-2988.1666
C01627=34.135,93.972,17.585,-179.9985,0.0798,-2989.9634
C01628=36.917,92.934,17.598,-179.9968,0.0074,-2991.6649
C01629=39.610,91.818,17.598,-179.9970,0.0075,-2993.3352
C01630=42.311,90.585,17.585,179.9996,0.0820,-2995.0366
C01631=45.077,89.109,17.565,-179.9709,0.3614,-2996.8332
C01632=47.692,87.339,17.545,-179.7213,1.8693,-2998.6370
C01633=49.816,85.535,17.521,-178.9354,4.2497,-3000.2167
C01634=51.202,83.948,17.473,-177.1153,6.7838,-3001.3801
C01635=52.143,82.495,17.374,-174.7815,10.0525,-3002.2959
C01636=53.070,81.058,17.237,-173.5629,15.1731,-3003.2134
C01637=54.382,79.482,17.095,-174.9324,20.6601,-3004.3801
C01638=56.571,77.464,16.986,-178.0125,24.0591,-3006.1402
C01639=60.019,74.640,16.941,-179.6996,25.0675,-3008.8032
C01640=63.789,71.434,16.939,179.9729,25.1255,-3011.7642
C01641=67.721,67.721,16.941,-180.0000,25.1124,-3015.0000
C01642=71.434,63.789,16.939,-179.9729,25.1255,-3018.2358
C01643=74.640,60.019,16.941,179.6996,25.0675,-3021.1968
C01644=77.464,56.571,16.986,178.0125,24.0591,-3023.8598
C01645=79.482,54.382,17.095,174.9324,20.6601,-3025.6199
C01646=81.058,53.070,17.237,173.5629,15.1731,-3026.7866
C01647=82.495,52.143,17.374,174.7815,10.0525,-3027.7041
C01648=83.948,51.202,17.473,177.1153,6.7838,-3028.6199
C01649=85.535,49.816,17.521,178.9354,4.2497,-3029.7833
C01650=87.339,47.692,17.545,179.7213,1.8693,-3031.3630
C01651=89.109,45.077,17.565,179.9709,0.3614,-3033.1668
C01652=90.585,42.311,17.585,-179.9996,0.0820,-3034.9634
C01653=91.818,39.610,17.598,179.9970,0.0075,-3036.6648
C01654=92.934,36.917,17.598,179.9968,0.0074,-3038.3351
C01655=93.972,34.135,17.585,179.9985,0.0798,-3040.0366
C01656=94.884,31.135,17.565,-179.9727,0.3589,-3041.8334
C01657=95.481,28.035,17.545,-179.7194,1.8706,-3043.6368
C01658=95.708,25.257,17.521,-178.9370,4.2461,-3045.2169
C01659=95.565,23.155,17.473,-177.1151,6.7819,-3046.3800
C01660=95.203,21.462,17.374,-174.7852,10.0480,-3047.2959
C01661=94.842,19.790,17.237,-173.5645,15.1715,-3048.2136
C01662=94.656,17.748,17.095,-174.9374,20.6589,-3049.3803
C01663=94.777,14.774,16.986,-178.0084,24.0583,-3051.1399
C01664=95.219,10.339,16.941,-179.6989,25.0665,-3053.8030
C01665=95.617,5.406,16.939,179.9726,25.1250,-3056.7641
C01666=95.772,0.000,16.941,180.0000,25.1121,-3060.0000
C01667=95.617,-5.406,16.939,-179.9726,25.1250,-3063.2359
C01668=95.219,-10.339,16.941,179.6989,25.0665,-3066.1970
C01669=94.777,-14.774,16.986,178.0146,24.0591,-3068.8601
C01670=94.656,-17.748,17.095,174.9374,20.6589,-3070.6197
C01671=94.842,-19.790,17.237,173.5645,15.1715,-3071.7864
C01672=95.203,-21.462,17.374,174.7852,10.0480,-3072.7041
C01673=95.565,-23.155,17.473,177.1151,6.7819,-3073.6200
C01674=95.708,-25.257,17.521,178.9370,4.2461,-3074.7831
C01675=95.481,-28.035,17.545,179.7194,1.8706,-3076.3632
C01676=94.884,-31.135,17.565,179.9727,0.3589,-3078.1666
C01677=93.972,-34.135,17.585,-179.9985,0.0798,-3079.9634
C01678=92.934,-36.917,17.598,-179.9968,0.0074,-3081.6649
C01679=91.818,-39.610,17.598,-179.9970,0.0075,-3083.3352
C01680=90.585,-42.311,17.585,179.9996,0.0820,-3085.0366
C01681=89.109,-45.077,17.565,-179.9709,0.3614,-3086.8332
C01682=87.339,-47.692,17.545,-179.7213,1.8693,-3088.6370
C01683=85.535,-49.816,17.521,-178.9354,4.2497,-3090.2167
C01684=83.948,-51.202,17.473,-177.1153,6.7838,-3091.3801
C01685=82.495,-52.143,17.374,-174.7815,10.0525,-3092.2959
C01686=81.058,-53.070,17.237,-173.5629,15.1731,-3093.2134
C01687=79.482,-54.382,17.095,-174.9324,20.6601,-3094.3801
C01688=77.464,-56.571,16.986,-178.0125,24.0591,-3096.1402
C01689=74.640,-60.019,16.941,-179.6996,25.0675,-3098.8032
C01690=71.434,-63.789,16.939,179.9729,25.1255,-3101.7642
C01691=67.721,-67.721,16.941,-180.0000,25.1124,-3105.0000
C01692=63.789,-71.434,16.939,-179.9729,25.1255,-3108.2358
C01693=60.019,-74.640,16.941,179.6996,25.0675,-3111.1968
C01694=56.571,-77.464,16.986,178.0125,24.0591,-3113.8598
C01695=54.382,-79.482,17.095,174.9324,20.6601,-3115.6199
C01696=53.070,-81.058,17.237,173.5629,15.1731,-3116.7866
C01697=52.143,-82.495,17.374,174.7815,10.0525,-3117.7041
C01698=51.202,-83.948,17.473,177.1153,6.7838,-3118.6199
C01699=49.816,-85.535,17.521,178.9354,4.2497,-3119.7833
C01700=47.692,-87.339,17.545,179.7213,1.8693,-3121.3630
C01701=45.077,-89.109,17.565,179.9709,0.3614,-3123.1668
C01702=42.311,-90.585,17.585,-179.9996,0.0820,-3124.9634
C01703=39.610,-91.818,17.598,179.9970,0.0075,-3126.6648
C01704=36.917,-92.934,17.598,179.9968,0.0074,-3128.3351
C01705=34.135,-93.972,17.585,179.9985,0.0798,-3130.0366
C01706=31.135,-94.884,17.565,-179.9727,0.3589,-3131.8334
C01707=28.035,-95.481,17.545,-179.7194,1.8706,-3133.6368
C01708=25.257,-95.708,17.521,-178.9370,4.2461,-3135.2169
C01709=23.155,-95.565,17.473,-177.1151,6.7819,-3136.3800
C01710=21.462,-95.203,17.374,-174.7852,10.0480,-3137.2959
C01711=19.790,-94.842,17.237,-173.5645,15.1715,-3138.2136
C01712=17.748,-94.656,17.095,-174.9374,20.6589,-3139.3803
C01713=14.774,-94.777,16.986,-178.0084,24.0583,-3141.1399
C01714=10.339,-95.219,16.941,-179.6989,25.0665,-3143.8030
C01715=5.406,-95.617,16.939,179.9726,25.1250,-3146.7641
C01716=0.000,-95.772,16.941,-180.0000,25.1121,-3150.0000
C01717=0.000,-95.772,16.941,-180.0000,25.1121,-3150.0000
C01718=-5.406,-95.617,16.939,-179.9726,25.1250,-3153.2359
C01719=-10.339,-95.219,16.941,179.6989,25.0665,-3156.1970
C01720=-14.774,-94.777,16.986,178.0146,24.0591,-3158.8601
C01721=-17.748,-94.656,17.095,174.9374,20.6589,-3160.6197
C01722=-19.790,-94.842,17.237,173.5645,15.1715,-3161.7864
C01723=-21.462,-95.203,17.374,174.7852,10.0480,-3162.7041
C01724=-23.155,-95.565,17.473,177.1151,6.7819,-3163.6200
C01725=-25.257,-95.708,17.521,178.9370,4.2461,-3164.7831
C01726=-28.035,-95.481,17.545,179.7194,1.8706,-3166.3632
C01727=-31.135,-94.884,17.565,179.9727,0.3589,-3168.1666
C01728=-34.135,-93.972,17.585,-179.9985,0.0798,-3169.9634
C01729=-36.917,-92.934,17.598,-179.9968,0.0074,-3171.6649
C01730=-39.610,-91.818,17.598,-179.9970,0.0075,-3173.3352
C01731=-42.311,-90.585,17.585,179.9996,0.0820,-3175.0366
C01732=-45.077,-89.109,17.565,-179.9709,0.3614,-3176.8332
C01733=-47.692,-87.339,17.545,-179.7213,1.8693,-3178.6370
C01734=-49.816,-85.535,17.521,-178.9354,4.2497,-3180.2167
C01735=-51.202,-83.948,17.473,-177.1153,6.7838,-3181.3801
C01736=-52.143,-82.495,17.374,-174.7815,10.0525,-3182.2959
C01737=-53.070,-81.058,17.237,-173.5629,15.1731,-3183.2134
C01738=-54.382,-79.482,17.095,-174.9324,20.6601,-3184.3801
C01739=-56.571,-77.464,16.986,-178.0125,24.0591,-3186.1402
C01740=-60.019,-74.640,16.941,-179.6996,25.0675,-3188.8032
C01741=-63.789,-71.434,16.939,179.9729,25.1255,-3191.7642
C01742=-67.721,-67.721,16.941,180.0000,25.1124,-3195.0000
C01743=-71.434,-63.789,16.939,-179.9729,25.1255,-3198.2358
C01744=-74.640,-60.019,16.941,179.6996,25.0675,-3201.1968
C01745=-77.464,-56.571,16.986,178.0125,24.0591,-3203.8598
C01746=-79.482,-54.382,17.095,174.9324,20.6601,-3205.6199
C01747=-81.058,-53.070,17.237,173.5629,15.1731,-3206.7866
C01748=-82.495,-52.143,17.374,174.7815,10.0525,-3207.7041
C01749=-83.948,-51.202,17.473,177.1153,6.7838,-3208.6199
C01750=-85.535,-49.816,17.521,178.9354,4.2497,-3209.7833
C01751=-87.339,-47.692,17.545,179.7213,1.8693,-3211.3630
C01752=-89.109,-45.077,17.565,179.9709,0.3614,-3213.1668
C01753=-90.585,-42.311,17.585,-179.9996,0.0820,-3214.9634
C01754=-91.818,-39.610,17.598,179.9970,0.0075,-3216.6648
C01755=-92.934,-36.917,17.598,179.9968,0.0074,-3218.3351
C01756=-93.972,-34.135,17.585,179.9985,0.0798,-3220.0366
C01757=-94.884,-31.135,17.565,-179.9727,0.3589,-3221.8334
C01758=-95.481,-28.035,17.545,-179.7194,1.8706,-3223.6368
C01759=-95.708,-25.257,17.521,-178.9370,4.2461,-3225.2169
C01760=-95.565,-23.155,17.473,-177.1151,6.7819,-3226.3800
C01761=-95.203,-21.462,17.374,-174.7852,10.0480,-3227.2959
C01762=-94.842,-19.790,17.237,-173.5645,15.1715,-3228.2136
C01763=-94.656,-17.748,17.095,-174.9374,20.6589,-3229.3803
C01764=-94.777,-14.774,16.986,-178.0084,24.0583,-3231.1399
C01765=-95.219,-10.339,16.941,-179.6989,25.0665,-3233.8030
C01766=-95.617,-5.406,16.939,179.9726,25.1250,-3236.7641
C01767=-95.772,0.000,16.941,-180.0000,25.1121,-3240.0000
C01768=-95.617,5.406,16.939,-179.9726,25.1250,-3243.2359
C01769=-95.219,10.339,16.941,179.6989,25.0665,-3246.1970
C01770=-94.777,14.774,16.986,178.0146,24.0591,-3248.8601
C01771=-94.656,17.748,17.095,174.9374,20.6589,-3250.6197
C01772=-94.842,19.790,17.237,173.5645,15.1715,-3251.7864
C01773=-95.203,21.462,17.374,174.7852,10.0480,-3252.7041
C01774=-95.565,23.155,17.473,177.1151,6.7819,-3253.6200
C01775=-95.708,25.257,17.521,178.9370,4.2461,-3254.7831
C01776=-95.481,28.035,17.545,179.7194,1.8706,-3256.3632
C01777=-94.884,31.135,17.565,179.9727,0.3589,-3258.1666
C01778=-93.972,34.135,17.585,-179.9985,0.0798,-3259.9634
C01779=-92.934,36.917,17.598,-179.9968,0.0074,-3261.6649
